// TIA Portal project "A180648-11总成异响" (V14)

(* hardware
DEVICE "S7-1200 station_1"  S7-1200 Station
   slot 0: "Rack_0"  S7-1200 Rack  Rack  V1.0
   slot 1: "A170648_14 CPU  1214C"  CPU 1214C DC/DC/DC  6ES7 214-1AG40-0XB0  V4.2
   slot 2: "DI 16/DQ 16x24VDC_1"  6ES7 223-1BL32-0XB0  V2.0
DEVICE "GSD device_1"  GSD.Device.PN
   slot 0: "机架"  Rack  V1.0
   slot 0: "cv-x100"  CV-X1XX  CV-X1XX  2.0
      slot 0: "CV-X1XX"  CV-X1XX  2.0
      slot 1: "Interface"  Interface
         slot 1: "Port 1"  Port 1
   slot 1: "Command and Result Status_1"  Command and Result Status
      slot 0: "Command and Result Status"  Command and Result Status
   slot 2: "Trg Ready Status_1"  Trg Ready Status
      slot 0: "Trg Ready Status"  Trg Ready Status
   slot 3: "Trg Ack Status_1"  Trg Ack Status
      slot 0: "Trg Ack Status"  Trg Ack Status
   slot 4: "Miscellaneous Status_1"  Miscellaneous Status
      slot 0: "Miscellaneous Status"  Miscellaneous Status
   slot 5: "Tool Judge Value_1"  Tool Judge Value
      slot 0: "Tool Judge Value"  Tool Judge Value
   slot 6: "Result Data 128Byte_1"  Result Data 128Byte
      slot 0: "Result Data 128Byte"  Result Data 128Byte
   slot 7: "Result Data 32Byte_1"  Result Data 32Byte
      slot 0: "Result Data 32Byte"  Result Data 32Byte
   slot 8: "Result Data 32Byte_2"  Result Data 32Byte
      slot 0: "Result Data 32Byte"  Result Data 32Byte
   slot 9: "Result Data 32Byte_3"  Result Data 32Byte
      slot 0: "Result Data 32Byte"  Result Data 32Byte
   slot 10: "Result Data 32Byte_4"  Result Data 32Byte
      slot 0: "Result Data 32Byte"  Result Data 32Byte
   slot 11: "Result Data 32Byte_5"  Result Data 32Byte
      slot 0: "Result Data 32Byte"  Result Data 32Byte
   slot 12: "Command and Result Control_1"  Command and Result Control
      slot 0: "Command and Result Control"  Command and Result Control
   slot 13: "Trg Control_1"  Trg Control
      slot 0: "Trg Control"  Trg Control
   slot 14: "Miscellaneous Control_1"  Miscellaneous Control
      slot 0: "Miscellaneous Control"  Miscellaneous Control
   slot 15: "Reserved Control_1"  Reserved Control
      slot 0: "Reserved Control"  Reserved Control
   slot 16: "Reserved Control_2"  Reserved Control
      slot 0: "Reserved Control"  Reserved Control
   slot 17: "Parameter 128Byte_1"  Parameter 128Byte
      slot 0: "Parameter 128Byte"  Parameter 128Byte
   slot 18: "Parameter 32Byte_1"  Parameter 32Byte
      slot 0: "Parameter 32Byte"  Parameter 32Byte
   slot 19: "Parameter 32Byte_2"  Parameter 32Byte
      slot 0: "Parameter 32Byte"  Parameter 32Byte
   slot 20: "Parameter 32Byte_3"  Parameter 32Byte
      slot 0: "Parameter 32Byte"  Parameter 32Byte
   slot 21: "Parameter 32Byte_4"  Parameter 32Byte
      slot 0: "Parameter 32Byte"  Parameter 32Byte
   slot 22: "Parameter 32Byte_5"  Parameter 32Byte
      slot 0: "Parameter 32Byte"  Parameter 32Byte
*)

// ===== PLC "A170648_14 CPU  1214C"  CPU 1214C DC/DC/DC =====

VAR_GLOBAL   // PLC tag table "默认变量表"
   "启动拍照" AT %I0.0 : Bool;
   "不" AT %I0.1 : Bool;
   "复位" AT %I0.2 : Bool;
   "急停" AT %I0.3 : Bool;
   "Tag_18" AT %IW64 : Int;
   "CMD_complete" AT %I504.0 : Bool;
   "TRG1_feed" AT %I506.0 : Bool;
   "TRG2_feed" AT %I506.1 : Bool;
   "CCD_busy" AT %I507.0 : Bool;
   "CCD_TRG1_NG" AT %I508.0 : Bool;
   "CCD_TRG1_OK" AT %I508.1 : Bool;
   "Conmmad Result" AT %ID588 : DWord;
   "Conmmad Data1" AT %ID592 : DWord;
   "Conmmad Data2" AT %ID596 : DWord;
   "电机拧紧确认" AT %I0.4 : Bool;
   "电机螺栓色标" AT %I3.7 : Bool;
   "电机扎带拾取" AT %I1.1 : Bool;
   "电机扫码启动" AT %I1.2 : Bool;
   "控制器扫码启动" AT %I2.0 : Bool;
   "拧紧枪2确认" AT %I0.5 : Bool;
   "拧紧枪3" AT %I0.6 : Bool;
   "ECU记号笔" AT %I1.5 : Bool;
   "左线卡" AT %I2.2 : Bool;
   "左轧带" AT %I2.5 : Bool;
   "Tag_27" AT %I0.7 : Bool;
   "中轧带" AT %I2.3 : Bool;
   "弹簧取料" AT %I2.4 : Bool;
   "红" AT %Q2.4 : Bool;
   "Tag_17" AT %QW80 : Int;
   "Tag_21" AT %Q3.2 : Bool;
   "Cmd Command" AT %Q504.0 : Bool;
   "CCD_reset" AT %Q504.4 : Bool;
   "TRG1.OUT" AT %Q505.0 : Bool;
   "TRG2.OUT" AT %Q505.1 : Bool;
   "RESET.OUT" AT %Q506.0 : Bool;
   "Tag_65" AT %Q506.1 : Bool;
   "Command NO.OUT" AT %QD580 : DWord;
   "Cmd Parameter1.OUT" AT %QD584 : DWord;
   "Cmd Parameter2.OUT" AT %QD588 : DWord;
   "Cmd Parameter3.OUT" AT %QD592 : DWord;
   "Cmd Parameter4.OUT" AT %QD596 : DWord;
   "Cmd Parameter5.OUT" AT %QD600 : DWord;
   "蜂鸣器" AT %Q2.3 : Bool;
   "Tag_42" AT %Q2.5 : Bool;
   "Tag_43" AT %Q2.6 : Bool;
   "Tag_44" AT %Q2.2 : Bool;
   "安装弹簧" AT %Q20.0 : Bool;
   "安装O型圈" AT %Q20.1 : Bool;
   "安装弹性垫圈弹簧" AT %Q20.2 : Bool;
   "电机安装螺栓1" AT %Q20.3 : Bool;
   "电机安装螺栓2" AT %Q20.4 : Bool;
   "电机安装螺栓3" AT %Q20.5 : Bool;
   "电机拍照" AT %Q20.6 : Bool;
   "涂色标" AT %Q20.7 : Bool;
   "安装轧带取走工" AT %Q21.0 : Bool;
   "Q29" AT %Q21.1 : Bool;
   "Q30" AT %Q21.2 : Bool;
   "Q31" AT %Q21.3 : Bool;
   "Q32" AT %Q21.4 : Bool;
   "Q33" AT %Q21.5 : Bool;
   "Q34" AT %Q21.6 : Bool;
   "Q35" AT %Q21.7 : Bool;
   "程序停止" AT %M100.0 : Bool;
   "复位完成" AT %M100.1 : Bool;
   "Clock_1Hz" AT %M0.5 : Bool;
   "AlwaysFALSE" AT %M1.3 : Bool;
   "Clock_Byte" AT %MB0 : Byte;
   "Clock_10Hz" AT %M0.0 : Bool;
   "Clock_5Hz" AT %M0.1 : Bool;
   "Clock_2.5Hz" AT %M0.2 : Bool;
   "Clock_2Hz" AT %M0.3 : Bool;
   "Clock_1.25Hz" AT %M0.4 : Bool;
   "Clock_0.625Hz" AT %M0.6 : Bool;
   "Clock_0.5Hz" AT %M0.7 : Bool;
   "System_Byte" AT %MB1 : Byte;
   "FirstScan" AT %M1.0 : Bool;
   "DiagStatusUpdate" AT %M1.1 : Bool;
   "AlwaysTRUE" AT %M1.2 : Bool;
   "Tag_19" AT %MD200 : Real;
   "Tag_20" AT %MD204 : Real;
   "磁粉离合器校准" AT %M160.0 : Bool;
   "Tag_22" AT %M300.1 : Bool;
   "Tag_23" AT %M300.2 : Bool;
   "Tag_24" AT %M300.3 : Bool;
   "Tag_25" AT %MW200 : Int;
   "Tag_26" AT %M400.0 : Bool;
   "Tag_1" AT %M200.0 : Bool;
   "Tag_2" AT %M200.1 : Bool;
   "Tag_3" AT %M200.2 : Bool;
   "Tag_4" AT %M200.3 : Bool;
   "Tag_5" AT %M200.4 : Bool;
   "Tag_6" AT %M200.5 : Bool;
   "Tag_7" AT %M200.6 : Bool;
   "Tag_8" AT %M200.7 : Bool;
   "Tag_9" AT %M201.0 : Bool;
   "Tag_10" AT %M201.1 : Bool;
   "Tag_11" AT %M201.2 : Bool;
   "Tag_12" AT %M201.3 : Bool;
   "Tag_13" AT %M201.4 : Bool;
   "Tag_14" AT %M201.5 : Bool;
   "Tag_15" AT %M201.6 : Bool;
   "Tag_16" AT %M201.7 : Bool;
   "Tag_17(1)" AT %M202.0 : Bool;
   "Tag_18(1)" AT %M202.1 : Bool;
   "Tag_19(1)" AT %M202.2 : Bool;
   "Tag_20(1)" AT %M202.3 : Bool;
   "Tag_21(1)" AT %M202.4 : Bool;
   "Tag_22(1)" AT %M202.5 : Bool;
   "Tag_23(1)" AT %M202.6 : Bool;
   "Tag_24(1)" AT %M202.7 : Bool;
   "Tag_37" AT %M203.0 : Bool;
   "Tag_38" AT %M203.1 : Bool;
   "Tag_39" AT %M203.2 : Bool;
   "Tag_40" AT %M205.0 : Bool;
   "Tag_41" AT %M205.1 : Bool;
   "Tag_45" AT %MW600 : Int;
   "Tag_46" AT %M500.0 : Bool;
   "Tag_47" AT %M500.1 : Bool;
   "Tag_48" AT %MW604 : Word;
   "Tag_49" AT %MW608 : Int;
   "Tag_28" AT %M500.3 : Bool;
   "Tag_29" AT %M500.5 : Bool;
   "Tag_30" AT %M501.0 : Bool;
   "Tag_31" AT %M501.1 : Bool;
   "Tag_32" AT %M503.0 : Bool;
   "Tag_33" AT %M503.1 : Bool;
   "Tag_34" AT %M503.2 : Bool;
   "Tag_35" AT %M503.3 : Bool;
   "Tag_36" AT %M503.4 : Bool;
   "Tag_50" AT %M503.5 : Bool;
   "Tag_51" AT %M505.0 : Bool;
   "Tag_52" AT %M506.0 : Bool;
   "Tag_53" AT %M506.1 : Bool;
   "Tag_54" AT %M506.2 : Bool;
   "Tag_55" AT %M506.5 : Bool;
   "Tag_56" AT %M506.6 : Bool;
   "Tag_57" AT %M507.1 : Bool;
   "Tag_58" AT %M507.0 : Bool;
   "Tag_59" AT %M507.2 : Bool;
   "控制器安装螺栓1" AT %Q30.0 : Bool;
   "控制器安装螺栓2" AT %Q30.1 : Bool;
   "控制器安装螺栓3" AT %Q30.2 : Bool;
   "安装支架螺栓1" AT %Q30.3 : Bool;
   "安装支架螺栓2" AT %Q30.4 : Bool;
   "安装支架螺栓3" AT %Q30.5 : Bool;
   "安装支架螺栓4" AT %Q30.6 : Bool;
   "安装支架涂色标" AT %Q30.7 : Bool;
   "安装轧带取走工件" AT %Q31.0 : Bool;
   "备用" AT %Q31.1 : Bool;
   "备用_1" AT %Q31.2 : Bool;
   "备用_2" AT %Q31.3 : Bool;
   "备用_3" AT %Q31.4 : Bool;
   "备用_4" AT %Q31.5 : Bool;
   "备用_5" AT %Q31.6 : Bool;
   "备用_6" AT %Q31.7 : Bool;
   "Tag_60" AT %M507.3 : Bool;
   "Tag_61" AT %M507.4 : Bool;
   "Tag_62" AT %M507.5 : Bool;
   "Tag_63" AT %M507.6 : Bool;
   "Tag_64" AT %M507.7 : Bool;
   "Tag_66" AT %M508.0 : Bool;
   "Tag_67" AT %M508.1 : Bool;
   "Tag_68" AT %M508.2 : Bool;
   "Tag_69" AT %M508.3 : Bool;
   "Tag_70" AT %M508.4 : Bool;
   "Tag_71" AT %M508.5 : Bool;
   "Tag_72" AT %M508.6 : Bool;
   "Tag_73" AT %M508.7 : Bool;
END_VAR

DATA_BLOCK "SERVER"   // DB1
{ S7_Optimized_Access := 'FALSE' }
VERSION : 0.1
   VAR
      设备状态1 : Int := 0;
      设备状态2 : Int;
      设备状态3 : Int;
      产品型号 : Int := 0;
      错误代码 : Int := 0;
      生产结果 : Int := 0;
      设备编号 : Int := 0;
      产品标识 : Int;
      胶垫弹簧CCD程序号 : Int;
      电机方向程序号 : Int;
      电机螺栓数量 : Int;
      合装螺栓1数量 : Int;
      合装螺栓2数量 : Int;
      控制器螺栓数量 : Int;
      ECU安装 : Array[0..16] of Bool;
   END_VAR
BEGIN
END_DATA_BLOCK

DATA_BLOCK "MB_TCON"   // DB2
{ S7_Optimized_Access := 'FALSE' }
VERSION : 0.1
   VAR
      MB_TCON : TCON_IP_v4;
   END_VAR
BEGIN
   MB_TCON.InterfaceId := 64;
   MB_TCON.ID := 1;
   MB_TCON.LocalPort := 502;
   MB_TCON.RemoteAddress.ADDR[1] := 0;
   MB_TCON.RemoteAddress.ADDR[2] := 0;
   MB_TCON.RemoteAddress.ADDR[3] := 0;
   MB_TCON.RemoteAddress.ADDR[4] := 0;
END_DATA_BLOCK

DATA_BLOCK "RESET_DB"   // DB3
{ S7_Optimized_Access := 'TRUE' }
VERSION : 0.1
// stored: InstanceOfName RESET
"RESET"
BEGIN
END_DATA_BLOCK

DATA_BLOCK "ALARM_DB"   // DB4
{ S7_Optimized_Access := 'TRUE' }
VERSION : 0.1
// stored: InstanceOfName ALARM
"ALARM"
BEGIN
END_DATA_BLOCK

DATA_BLOCK "CCD检测_DB"   // DB6
{ S7_Optimized_Access := 'TRUE' }
VERSION : 0.1
// stored: InstanceOfName CCD检测
"CCD检测"
BEGIN
END_DATA_BLOCK

DATA_BLOCK "AUTO_DB"   // DB10
{ S7_Optimized_Access := 'TRUE' }
VERSION : 0.1
// stored: InstanceOfName AUTO
"AUTO"
BEGIN
END_DATA_BLOCK

// folder: System blocks/Program resources

DATA_BLOCK "IEC_Timer_0_DB"   // DB5
{ S7_Optimized_Access := 'TRUE' }
AUTHOR : Simatic
FAMILY : IEC
NAME : IEC_TMR
VERSION : 1.0
// stored: InstanceOfName IEC_TIMER
"IEC_TIMER"
BEGIN
END_DATA_BLOCK

DATA_BLOCK "IEC_Timer_0_DB_3"   // DB12
{ S7_Optimized_Access := 'TRUE' }
AUTHOR : Simatic
FAMILY : IEC
NAME : IEC_TMR
VERSION : 1.0
// stored: InstanceOfName IEC_TIMER
"IEC_TIMER"
BEGIN
END_DATA_BLOCK

// folder: (top level)

FUNCTION_BLOCK "ALARM"   // FB1, LAD
{ S7_Optimized_Access := 'TRUE' }
VERSION : 0.1
   VAR
      "Error-ID" : Word;
      TEmp : Array[0..3] of Bool;
      IEC_Timer_0_Instance : TON_TIME;
      IEC_Timer_0_Instance_1 : TON_TIME;
      IEC_Timer_0_Instance_2 : TON_TIME;
      IEC_Timer_0_Instance_3 : TON_TIME;
      IEC_Timer_0_Instance_4 : TON_TIME;
      IEC_Timer_0_Instance_5 : TON_TIME;
      IEC_Timer_0_Instance_6 : TON_TIME;
      IEC_Timer_0_Instance_7 : TON_TIME;
      IEC_Timer_0_Instance_8 : TON_TIME;
      IEC_Timer_0_Instance_9 : TON_TIME;
      IEC_Timer_0_Instance_10 : TON_TIME;
      IEC_Timer_0_Instance_11 : TON_TIME;
      IEC_Timer_0_Instance_12 : TON_TIME;
      IEC_Timer_0_Instance_13 : TON_TIME;
      IEC_Timer_0_Instance_14 : TON_TIME;
      "STEP" : Int;
      IEC_Timer_0_Instance_15 : TON_TIME;
      IEC_Timer_0_Instance_16 : TON_TIME;
   END_VAR
BEGIN

REGION Network 1
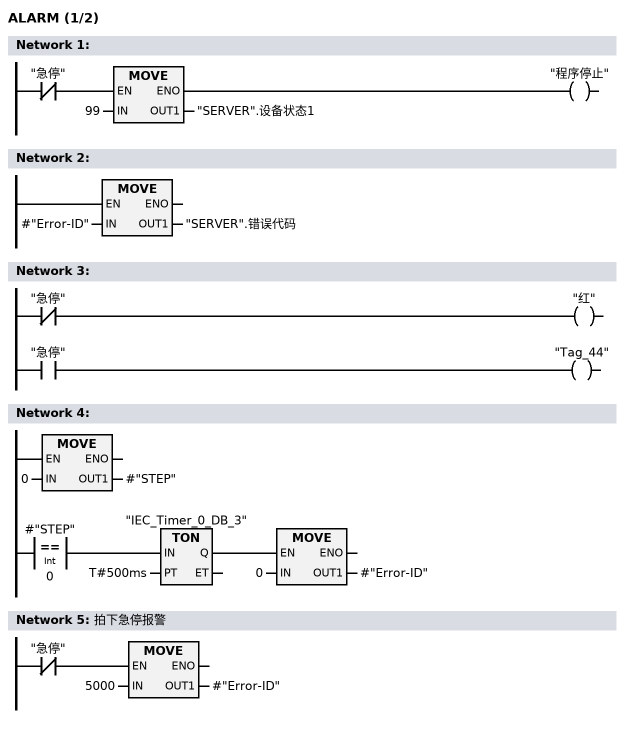
   RUNG wire#powerrail
      I_Contact( "急停" )
      Move(in := 99, out1 => "SERVER".设备状态1)
      Coil( "程序停止" )
   END_RUNG
   // the same network as SCL:
   IF NOT "急停" THEN "SERVER".设备状态1 := 99; END_IF;
   "程序停止" := NOT "急停";
END_REGION

REGION Network 2
   RUNG wire#powerrail
      Move(in := #"Error-ID", out1 => "SERVER".错误代码)
   END_RUNG
   // the same network as SCL:
   "SERVER".错误代码 := #"Error-ID";
END_REGION

REGION Network 3
   RUNG wire#powerrail
      I_Contact( "急停" )
      Coil( "红" )
   END_RUNG
   RUNG wire#powerrail
      Contact( "急停" )
      Coil( "Tag_44" )
   END_RUNG
   // the same network as SCL:
   "红" := NOT "急停";
   "Tag_44" := "急停";
END_REGION

REGION Network 4
   #"STEP" := 0;
   "IEC_Timer_0_DB_3".TON(IN := #"STEP" = 0, PT := T#500ms);
   IF "IEC_Timer_0_DB_3".Q THEN #"Error-ID" := 0; END_IF;
END_REGION

REGION Network 5: 拍下急停报警
   RUNG wire#powerrail
      I_Contact( "急停" )
      Move(in := 5000, out1 => #"Error-ID")
   END_RUNG
   // the same network as SCL:
   IF NOT "急停" THEN #"Error-ID" := 5000; END_IF;
END_REGION

REGION Network 6: 安全门打开报警
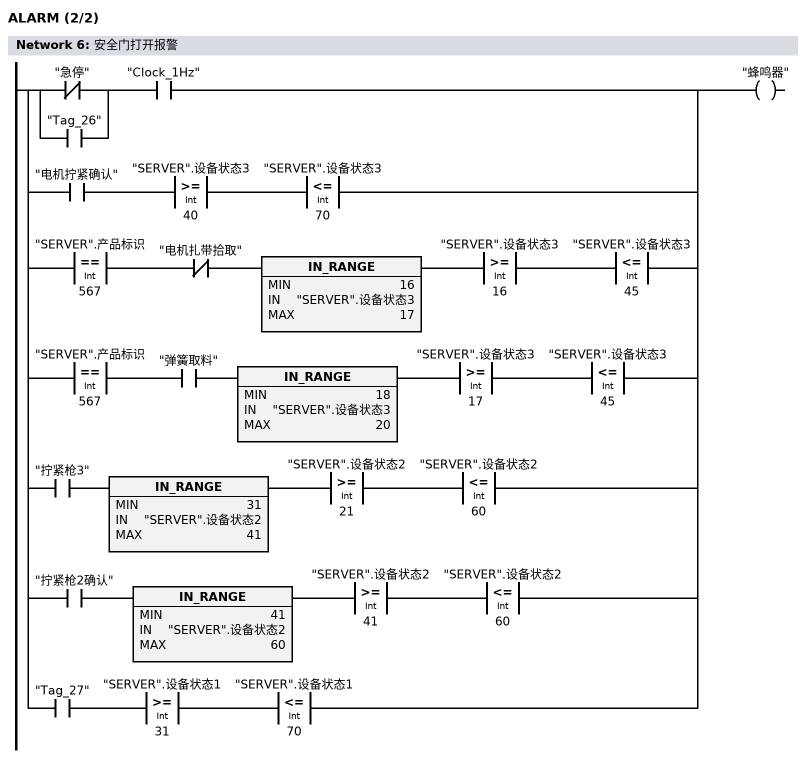
   RUNG wire#powerrail
      I_Contact( "急停" )
      wire#w1
      Contact( "Clock_1Hz" )
      wire#w2
      Coil( "蜂鸣器" )
   END_RUNG
   RUNG wire#powerrail
      Contact( "Tag_26" )
   END_RUNG wire#w1
   RUNG wire#powerrail
      Contact( "电机拧紧确认" )
      { S7_Templates := "SrcType := Int" } GE_Contact(in1 := "SERVER".设备状态3, in2 := 40)
      { S7_Templates := "SrcType := Int" } LE_Contact(in1 := "SERVER".设备状态3, in2 := 70)
   END_RUNG wire#w2
   RUNG wire#powerrail
      { S7_Templates := "SrcType := Int" } EQ_Contact(in1 := "SERVER".产品标识, in2 := 567)
      I_Contact( "电机扎带拾取" )
      { S7_Templates := "SrcType := Int" } InRange(min := 16, in := "SERVER".设备状态3, max := 17)
      { S7_Templates := "SrcType := Int" } GE_Contact(in1 := "SERVER".设备状态3, in2 := 16)
      { S7_Templates := "SrcType := Int" } LE_Contact(in1 := "SERVER".设备状态3, in2 := 45)
   END_RUNG wire#w2
   RUNG wire#powerrail
      { S7_Templates := "SrcType := Int" } EQ_Contact(in1 := "SERVER".产品标识, in2 := 567)
      Contact( "弹簧取料" )
      { S7_Templates := "SrcType := Int" } InRange(min := 18, in := "SERVER".设备状态3, max := 20)
      { S7_Templates := "SrcType := Int" } GE_Contact(in1 := "SERVER".设备状态3, in2 := 17)
      { S7_Templates := "SrcType := Int" } LE_Contact(in1 := "SERVER".设备状态3, in2 := 45)
   END_RUNG wire#w2
   RUNG wire#powerrail
      Contact( "拧紧枪3" )
      { S7_Templates := "SrcType := Int" } InRange(min := 31, in := "SERVER".设备状态2, max := 41)
      { S7_Templates := "SrcType := Int" } GE_Contact(in1 := "SERVER".设备状态2, in2 := 21)
      { S7_Templates := "SrcType := Int" } LE_Contact(in1 := "SERVER".设备状态2, in2 := 60)
   END_RUNG wire#w2
   RUNG wire#powerrail
      Contact( "拧紧枪2确认" )
      { S7_Templates := "SrcType := Int" } InRange(min := 41, in := "SERVER".设备状态2, max := 60)
      { S7_Templates := "SrcType := Int" } GE_Contact(in1 := "SERVER".设备状态2, in2 := 41)
      { S7_Templates := "SrcType := Int" } LE_Contact(in1 := "SERVER".设备状态2, in2 := 60)
   END_RUNG wire#w2
   RUNG wire#powerrail
      Contact( "Tag_27" )
      { S7_Templates := "SrcType := Int" } GE_Contact(in1 := "SERVER".设备状态1, in2 := 31)
      { S7_Templates := "SrcType := Int" } LE_Contact(in1 := "SERVER".设备状态1, in2 := 70)
   END_RUNG wire#w2
   // the same network as SCL:
   "蜂鸣器" := ((NOT "急停" OR "Tag_26") AND "Clock_1Hz") OR ("电机拧紧确认" AND ("SERVER".设备状态3 >= 40) AND ("SERVER".设备状态3 <= 70)) OR (("SERVER".产品标识 = 567) AND NOT "电机扎带拾取" AND (16 <= "SERVER".设备状态3) AND ("SERVER".设备状态3 <= 17) AND ("SERVER".设备状态3 >= 16) AND ("SERVER".设备状态3 <= 45)) OR (("SERVER".产品标识 = 567) AND "弹簧取料" AND (18 <= "SERVER".设备状态3) AND ("SERVER".设备状态3 <= 20) AND ("SERVER".设备状态3 >= 17) AND ("SERVER".设备状态3 <= 45)) OR ("拧紧枪3" AND (31 <= "SERVER".设备状态2) AND ("SERVER".设备状态2 <= 41) AND ("SERVER".设备状态2 >= 21) AND ("SERVER".设备状态2 <= 60)) OR ("拧紧枪2确认" AND (41 <= "SERVER".设备状态2) AND ("SERVER".设备状态2 <= 60) AND ("SERVER".设备状态2 >= 41) AND ("SERVER".设备状态2 <= 60)) OR ("Tag_27" AND ("SERVER".设备状态1 >= 31) AND ("SERVER".设备状态1 <= 70));
END_REGION

REGION Network 7: 工件未在位启动报警
END_REGION

REGION Network 8: 气源未开报警
END_REGION

REGION Network 9: 工装移栽前进未到位报警
END_REGION

REGION Network 10: 工装移栽未后退报警
END_REGION

REGION Network 11: 防护门未上升报警
END_REGION

REGION Network 12: 防护门为下降报警
END_REGION

REGION Network 13: 1#固定气缸未锁紧报警
END_REGION

REGION Network 14: 1#固定气缸未退回报警
END_REGION

REGION Network 15: 1#机械手未上升报警
END_REGION

REGION Network 16: 1#机械手未下降报警
END_REGION

REGION Network 17: 1#气爪未夹紧到位报警
END_REGION

REGION Network 18: 1#气爪未松开报警
END_REGION

REGION Network 19: 2#机械手未固定锁紧报警
END_REGION

REGION Network 20: 2#固定气缸未退回报警
END_REGION

REGION Network 21: 2#机械手未上升报警
END_REGION

REGION Network 22: 2#机械手未下降报警
END_REGION

REGION Network 23: 2#气爪未夹紧报警
END_REGION

REGION Network 24: 2#气爪未松开报警
END_REGION

REGION Network 25: 激光打码报警
END_REGION
END_FUNCTION_BLOCK

FUNCTION_BLOCK "RESET"   // FB2, LAD
{ S7_Optimized_Access := 'TRUE' }
VERSION : 0.1
   VAR_INPUT
      Stop : Bool;
      Start : Bool;
   END_VAR
   VAR_OUTPUT
      Down : Bool;
   END_VAR
   VAR
      "Step" : Int;
   END_VAR
BEGIN

REGION Network 1
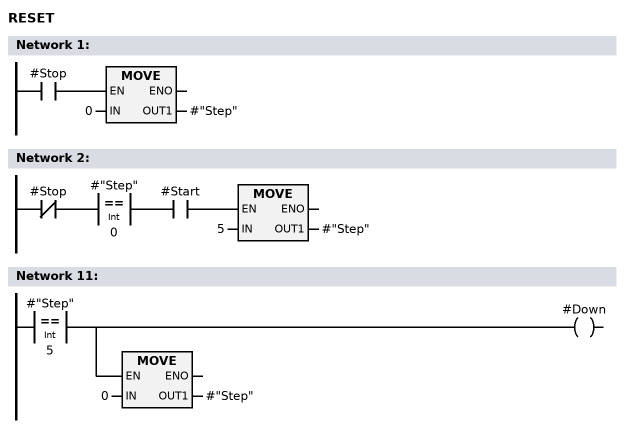
   RUNG wire#powerrail
      Contact( #Stop )
      Move(in := 0, out1 => #"Step")
   END_RUNG
   // the same network as SCL:
   IF #Stop THEN #"Step" := 0; END_IF;
END_REGION

REGION Network 2
   RUNG wire#powerrail
      I_Contact( #Stop )
      { S7_Templates := "SrcType := Int" } EQ_Contact(in1 := #"Step", in2 := 0)
      Contact( #Start )
      Move(in := 5, out1 => #"Step")
   END_RUNG
   // the same network as SCL:
   IF NOT #Stop AND (#"Step" = 0) AND #Start THEN #"Step" := 5; END_IF;
END_REGION

REGION Network 7: 1#气爪松开
END_REGION

REGION Network 8: 2#气爪松开
END_REGION

REGION Network 11
   RUNG wire#powerrail
      { S7_Templates := "SrcType := Int" } EQ_Contact(in1 := #"Step", in2 := 5)
      wire#w1
      Coil( #Down )
   END_RUNG
   RUNG wire#w1
      Move(in := 0, out1 => #"Step")
   END_RUNG
   // the same network as SCL:
   #Down := #"Step" = 5;
   IF #Down THEN #"Step" := 0; END_IF;
END_REGION
END_FUNCTION_BLOCK

FUNCTION_BLOCK "AUTO"   // FB3, LAD
{ S7_Optimized_Access := 'TRUE' }
VERSION : 0.1
   VAR
      IEC_Timer_0_Instance : TON_TIME;
      IEC_Timer_0_Instance_1 : TON_TIME;
      IEC_Timer_0_Instance_2 : TON_TIME;
      IEC_Timer_0_Instance_3 : TON_TIME;
      IEC_Timer_0_Instance_4 : TON_TIME;
      IEC_Timer_0_Instance_5 : TON_TIME;
      IEC_Timer_0_Instance_6 : TON_TIME;
      IEC_Timer_0_Instance_7 : TON_TIME;
      IEC_Timer_0_Instance_8 : TON_TIME;
      IEC_Timer_0_Instance_9 : TON_TIME;
      IEC_Timer_0_Instance_10 : TON_TIME;
      IEC_Timer_0_Instance_11 : TON_TIME;
      IEC_Timer_0_Instance_12 : TON_TIME;
      IEC_Timer_0_Instance_13 : TON_TIME;
      IEC_Timer_0_Instance_14 : TON_TIME;
      IEC_Timer_0_Instance_15 : TON_TIME;
      IEC_Timer_0_Instance_16 : TON_TIME;
      IEC_Timer_0_Instance_17 : TON_TIME;
      IEC_Timer_0_Instance_18 : TON_TIME;
      IEC_Timer_0_Instance_19 : TON_TIME;
      IEC_Timer_0_Instance_20 : TON_TIME;
      IEC_Timer_0_Instance_22 : TON_TIME;
      IEC_Timer_0_Instance_23 : TON_TIME;
      IEC_Timer_0_Instance_21 : TON_TIME;
   END_VAR
   VAR_TEMP
      temp0 : Bool;
      temp1 : Bool;
      temp2 : Bool;
      temp17 : Bool;
      temp4 : Bool;
      temp5 : Bool;
      temp6 : Bool;
      temp7 : Bool;
      temp8 : Bool;
      temp9 : Bool;
      temp10 : Bool;
      temp11 : Bool;
      temp12 : Bool;
      temp13 : Bool;
      temp14 : Bool;
      temp15 : Bool;
      temp16 : Bool;
      temp18 : Bool;
      temp19 : Bool;
      temp20 : Bool;
      temp21 : Bool;
   END_VAR
   VAR_TEMP   // added for the SCL form of the ladder/FBD networks
      _w1 : Bool;
      _w2 : Bool;
      _w3 : Bool;
      _w4 : Bool;
   END_VAR
BEGIN

REGION Network 1
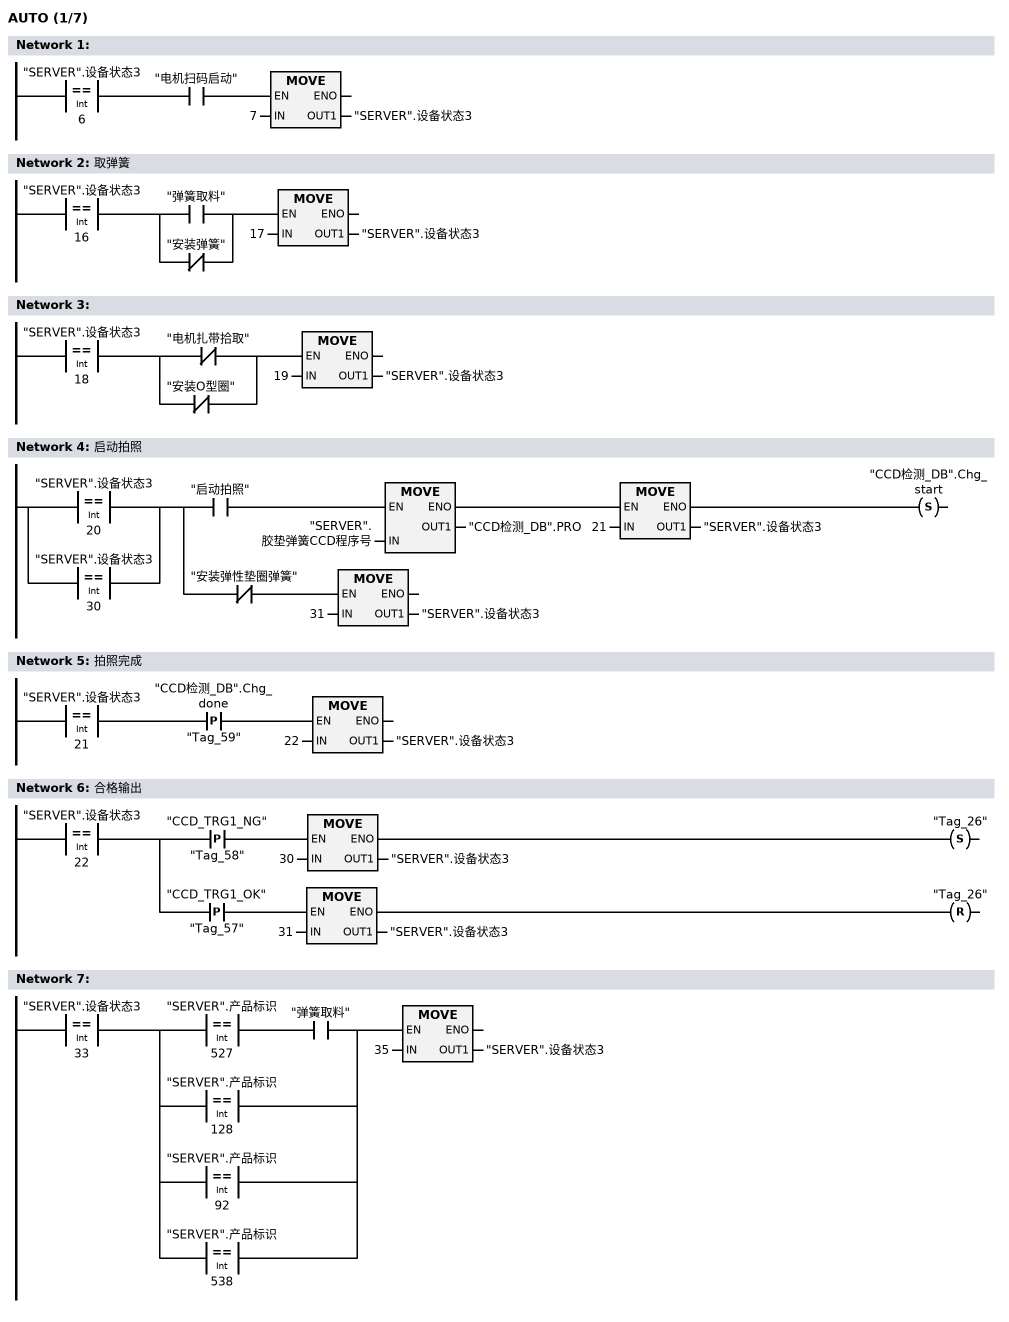
   RUNG wire#powerrail
      { S7_Templates := "SrcType := Int" } EQ_Contact(in1 := "SERVER".设备状态3, in2 := 6)
      Contact( "电机扫码启动" )
      Move(in := 7, out1 => "SERVER".设备状态3)
   END_RUNG
   // the same network as SCL:
   IF ("SERVER".设备状态3 = 6) AND "电机扫码启动" THEN "SERVER".设备状态3 := 7; END_IF;
END_REGION

REGION Network 2: 取弹簧
   RUNG wire#powerrail
      { S7_Templates := "SrcType := Int" } EQ_Contact(in1 := "SERVER".设备状态3, in2 := 16)
      wire#w1
      Contact( "弹簧取料" )
      wire#w2
      Move(in := 17, out1 => "SERVER".设备状态3)
   END_RUNG
   RUNG wire#w1
      I_Contact( "安装弹簧" )
   END_RUNG wire#w2
   // the same network as SCL:
   IF ("SERVER".设备状态3 = 16) AND ("弹簧取料" OR NOT "安装弹簧") THEN "SERVER".设备状态3 := 17; END_IF;
END_REGION

REGION Network 3
   RUNG wire#powerrail
      { S7_Templates := "SrcType := Int" } EQ_Contact(in1 := "SERVER".设备状态3, in2 := 18)
      wire#w1
      I_Contact( "电机扎带拾取" )
      wire#w2
      Move(in := 19, out1 => "SERVER".设备状态3)
   END_RUNG
   RUNG wire#w1
      I_Contact( "安装O型圈" )
   END_RUNG wire#w2
   // the same network as SCL:
   IF ("SERVER".设备状态3 = 18) AND (NOT "电机扎带拾取" OR NOT "安装O型圈") THEN "SERVER".设备状态3 := 19; END_IF;
END_REGION

REGION Network 4: 启动拍照
   RUNG wire#powerrail
      { S7_Templates := "SrcType := Int" } EQ_Contact(in1 := "SERVER".设备状态3, in2 := 20)
      wire#w1
      Contact( "启动拍照" )
      Move(in := "SERVER".胶垫弹簧CCD程序号, out1 => "CCD检测_DB".PRO)
      Move(in := 21, out1 => "SERVER".设备状态3)
      S_Coil( "CCD检测_DB".Chg_start )
   END_RUNG
   RUNG wire#powerrail
      { S7_Templates := "SrcType := Int" } EQ_Contact(in1 := "SERVER".设备状态3, in2 := 30)
   END_RUNG wire#w1
   RUNG wire#w1
      I_Contact( "安装弹性垫圈弹簧" )
      Move(in := 31, out1 => "SERVER".设备状态3)
   END_RUNG
   // the same network as SCL:
   #_w1 := ("SERVER".设备状态3 = 20) OR ("SERVER".设备状态3 = 30);
   IF #_w1 AND "启动拍照" THEN
       "CCD检测_DB".PRO := "SERVER".胶垫弹簧CCD程序号;
       "SERVER".设备状态3 := 21;
       "CCD检测_DB".Chg_start := TRUE;
   END_IF;
   IF #_w1 AND NOT "安装弹性垫圈弹簧" THEN "SERVER".设备状态3 := 31; END_IF;
END_REGION

REGION Network 5: 拍照完成
   RUNG wire#powerrail
      { S7_Templates := "SrcType := Int" } EQ_Contact(in1 := "SERVER".设备状态3, in2 := 21)
      P_Contact(operand := "CCD检测_DB".Chg_done, bit := "Tag_59")
      Move(in := 22, out1 => "SERVER".设备状态3)
   END_RUNG
   // the same network as SCL:
   #_w1 := ("SERVER".设备状态3 = 21) AND "CCD检测_DB".Chg_done AND NOT "Tag_59";   // rising edge of "CCD检测_DB".Chg_done
   "Tag_59" := "CCD检测_DB".Chg_done;
   IF #_w1 THEN "SERVER".设备状态3 := 22; END_IF;
END_REGION

REGION Network 6: 合格输出
   RUNG wire#powerrail
      { S7_Templates := "SrcType := Int" } EQ_Contact(in1 := "SERVER".设备状态3, in2 := 22)
      wire#w1
      P_Contact(operand := "CCD_TRG1_NG", bit := "Tag_58")
      Move(in := 30, out1 => "SERVER".设备状态3)
      S_Coil( "Tag_26" )
   END_RUNG
   RUNG wire#w1
      P_Contact(operand := "CCD_TRG1_OK", bit := "Tag_57")
      Move(in := 31, out1 => "SERVER".设备状态3)
      R_Coil( "Tag_26" )
   END_RUNG
   // the same network as SCL:
   #_w1 := "SERVER".设备状态3 = 22;
   #_w2 := #_w1 AND "CCD_TRG1_NG" AND NOT "Tag_58";   // rising edge of "CCD_TRG1_NG"
   "Tag_58" := "CCD_TRG1_NG";
   IF #_w2 THEN
       "SERVER".设备状态3 := 30;
       "Tag_26" := TRUE;
   END_IF;
   #_w3 := #_w1 AND "CCD_TRG1_OK" AND NOT "Tag_57";   // rising edge of "CCD_TRG1_OK"
   "Tag_57" := "CCD_TRG1_OK";
   IF #_w3 THEN
       "SERVER".设备状态3 := 31;
       "Tag_26" := FALSE;
   END_IF;
END_REGION

REGION Network 7
   RUNG wire#powerrail
      { S7_Templates := "SrcType := Int" } EQ_Contact(in1 := "SERVER".设备状态3, in2 := 33)
      wire#w1
      { S7_Templates := "SrcType := Int" } EQ_Contact(in1 := "SERVER".产品标识, in2 := 527)
      Contact( "弹簧取料" )
      wire#w2
      Move(in := 35, out1 => "SERVER".设备状态3)
   END_RUNG
   RUNG wire#w1
      { S7_Templates := "SrcType := Int" } EQ_Contact(in1 := "SERVER".产品标识, in2 := 128)
   END_RUNG wire#w2
   RUNG wire#w1
      { S7_Templates := "SrcType := Int" } EQ_Contact(in1 := "SERVER".产品标识, in2 := 92)
   END_RUNG wire#w2
   RUNG wire#w1
      { S7_Templates := "SrcType := Int" } EQ_Contact(in1 := "SERVER".产品标识, in2 := 538)
   END_RUNG wire#w2
   // the same network as SCL:
   IF ("SERVER".设备状态3 = 33) AND ((("SERVER".产品标识 = 527) AND "弹簧取料") OR ("SERVER".产品标识 = 128) OR ("SERVER".产品标识 = 92) OR ("SERVER".产品标识 = 538)) THEN
       "SERVER".设备状态3 := 35;
   END_IF;
END_REGION

REGION Network 8
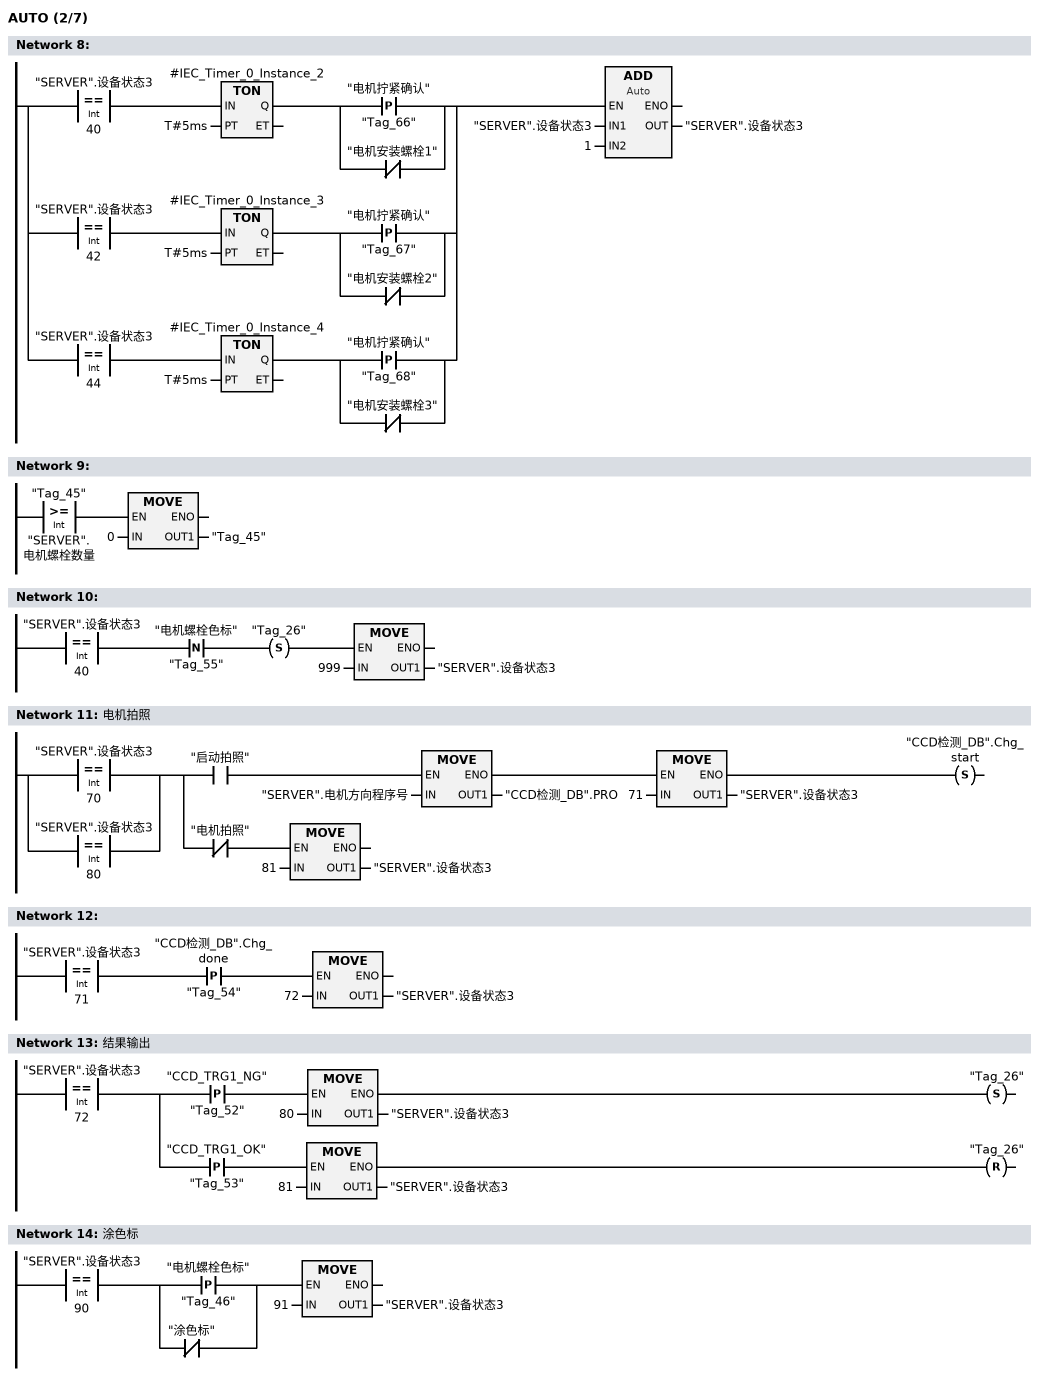
   #IEC_Timer_0_Instance_2(IN := "SERVER".设备状态3 = 40, PT := T#5ms);   // TON
   #_w1 := #IEC_Timer_0_Instance_2.Q AND "电机拧紧确认" AND NOT "Tag_66";   // rising edge of "电机拧紧确认"
   "Tag_66" := "电机拧紧确认";
   #IEC_Timer_0_Instance_3(IN := "SERVER".设备状态3 = 42, PT := T#5ms);   // TON
   #_w2 := #IEC_Timer_0_Instance_3.Q AND "电机拧紧确认" AND NOT "Tag_67";   // rising edge of "电机拧紧确认"
   "Tag_67" := "电机拧紧确认";
   #IEC_Timer_0_Instance_4(IN := "SERVER".设备状态3 = 44, PT := T#5ms);   // TON
   #_w3 := #IEC_Timer_0_Instance_4.Q AND "电机拧紧确认" AND NOT "Tag_68";   // rising edge of "电机拧紧确认"
   "Tag_68" := "电机拧紧确认";
   IF #_w1 OR (#IEC_Timer_0_Instance_2.Q AND NOT "电机安装螺栓1") OR #_w2 OR (#IEC_Timer_0_Instance_3.Q AND NOT "电机安装螺栓2") OR #_w3 OR (#IEC_Timer_0_Instance_4.Q AND NOT "电机安装螺栓3") THEN
       "SERVER".设备状态3 := "SERVER".设备状态3 + 1;
   END_IF;
END_REGION

REGION Network 9
   RUNG wire#powerrail
      { S7_Templates := "SrcType := Int" } GE_Contact(in1 := "Tag_45", in2 := "SERVER".电机螺栓数量)
      Move(in := 0, out1 => "Tag_45")
   END_RUNG
   // the same network as SCL:
   IF "Tag_45" >= "SERVER".电机螺栓数量 THEN "Tag_45" := 0; END_IF;
END_REGION

REGION Network 10
   RUNG wire#powerrail
      { S7_Templates := "SrcType := Int" } EQ_Contact(in1 := "SERVER".设备状态3, in2 := 40)
      N_Contact(operand := "电机螺栓色标", bit := "Tag_55")
      S_Coil( "Tag_26" )
      Move(in := 999, out1 => "SERVER".设备状态3)
   END_RUNG
   // the same network as SCL:
   #_w1 := ("SERVER".设备状态3 = 40) AND NOT "电机螺栓色标" AND "Tag_55";   // falling edge of "电机螺栓色标"
   "Tag_55" := "电机螺栓色标";
   IF #_w1 THEN
       "Tag_26" := TRUE;
       "SERVER".设备状态3 := 999;
   END_IF;
END_REGION

REGION Network 11: 电机拍照
   RUNG wire#powerrail
      { S7_Templates := "SrcType := Int" } EQ_Contact(in1 := "SERVER".设备状态3, in2 := 70)
      wire#w1
      Contact( "启动拍照" )
      Move(in := "SERVER".电机方向程序号, out1 => "CCD检测_DB".PRO)
      Move(in := 71, out1 => "SERVER".设备状态3)
      S_Coil( "CCD检测_DB".Chg_start )
   END_RUNG
   RUNG wire#powerrail
      { S7_Templates := "SrcType := Int" } EQ_Contact(in1 := "SERVER".设备状态3, in2 := 80)
   END_RUNG wire#w1
   RUNG wire#w1
      I_Contact( "电机拍照" )
      Move(in := 81, out1 => "SERVER".设备状态3)
   END_RUNG
   // the same network as SCL:
   #_w1 := ("SERVER".设备状态3 = 70) OR ("SERVER".设备状态3 = 80);
   IF #_w1 AND "启动拍照" THEN
       "CCD检测_DB".PRO := "SERVER".电机方向程序号;
       "SERVER".设备状态3 := 71;
       "CCD检测_DB".Chg_start := TRUE;
   END_IF;
   IF #_w1 AND NOT "电机拍照" THEN "SERVER".设备状态3 := 81; END_IF;
END_REGION

REGION Network 12
   RUNG wire#powerrail
      { S7_Templates := "SrcType := Int" } EQ_Contact(in1 := "SERVER".设备状态3, in2 := 71)
      P_Contact(operand := "CCD检测_DB".Chg_done, bit := "Tag_54")
      Move(in := 72, out1 => "SERVER".设备状态3)
   END_RUNG
   // the same network as SCL:
   #_w1 := ("SERVER".设备状态3 = 71) AND "CCD检测_DB".Chg_done AND NOT "Tag_54";   // rising edge of "CCD检测_DB".Chg_done
   "Tag_54" := "CCD检测_DB".Chg_done;
   IF #_w1 THEN "SERVER".设备状态3 := 72; END_IF;
END_REGION

REGION Network 13: 结果输出
   RUNG wire#powerrail
      { S7_Templates := "SrcType := Int" } EQ_Contact(in1 := "SERVER".设备状态3, in2 := 72)
      wire#w1
      P_Contact(operand := "CCD_TRG1_NG", bit := "Tag_52")
      Move(in := 80, out1 => "SERVER".设备状态3)
      S_Coil( "Tag_26" )
   END_RUNG
   RUNG wire#w1
      P_Contact(operand := "CCD_TRG1_OK", bit := "Tag_53")
      Move(in := 81, out1 => "SERVER".设备状态3)
      R_Coil( "Tag_26" )
   END_RUNG
   // the same network as SCL:
   #_w1 := "SERVER".设备状态3 = 72;
   #_w2 := #_w1 AND "CCD_TRG1_NG" AND NOT "Tag_52";   // rising edge of "CCD_TRG1_NG"
   "Tag_52" := "CCD_TRG1_NG";
   IF #_w2 THEN
       "SERVER".设备状态3 := 80;
       "Tag_26" := TRUE;
   END_IF;
   #_w3 := #_w1 AND "CCD_TRG1_OK" AND NOT "Tag_53";   // rising edge of "CCD_TRG1_OK"
   "Tag_53" := "CCD_TRG1_OK";
   IF #_w3 THEN
       "SERVER".设备状态3 := 81;
       "Tag_26" := FALSE;
   END_IF;
END_REGION

REGION Network 14: 涂色标
   RUNG wire#powerrail
      { S7_Templates := "SrcType := Int" } EQ_Contact(in1 := "SERVER".设备状态3, in2 := 90)
      wire#w1
      P_Contact(operand := "电机螺栓色标", bit := "Tag_46")
      wire#w2
      Move(in := 91, out1 => "SERVER".设备状态3)
   END_RUNG
   RUNG wire#w1
      I_Contact( "涂色标" )
   END_RUNG wire#w2
   // the same network as SCL:
   #_w1 := ("SERVER".设备状态3 = 90) AND "电机螺栓色标" AND NOT "Tag_46";   // rising edge of "电机螺栓色标"
   "Tag_46" := "电机螺栓色标";
   IF #_w1 OR (("SERVER".设备状态3 = 90) AND NOT "涂色标") THEN "SERVER".设备状态3 := 91; END_IF;
END_REGION

REGION Network 15
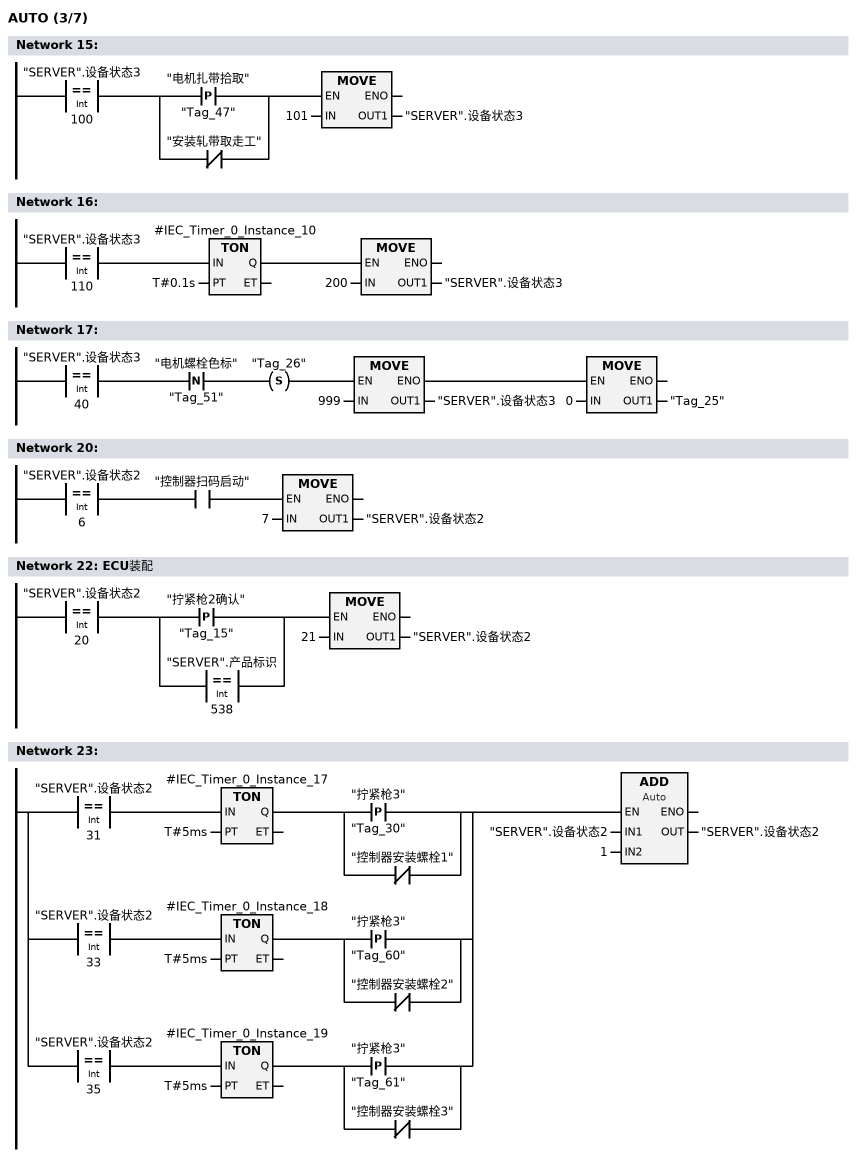
   RUNG wire#powerrail
      { S7_Templates := "SrcType := Int" } EQ_Contact(in1 := "SERVER".设备状态3, in2 := 100)
      wire#w1
      P_Contact(operand := "电机扎带拾取", bit := "Tag_47")
      wire#w2
      Move(in := 101, out1 => "SERVER".设备状态3)
   END_RUNG
   RUNG wire#w1
      I_Contact( "安装轧带取走工" )
   END_RUNG wire#w2
   // the same network as SCL:
   #_w1 := ("SERVER".设备状态3 = 100) AND "电机扎带拾取" AND NOT "Tag_47";   // rising edge of "电机扎带拾取"
   "Tag_47" := "电机扎带拾取";
   IF #_w1 OR (("SERVER".设备状态3 = 100) AND NOT "安装轧带取走工") THEN "SERVER".设备状态3 := 101; END_IF;
END_REGION

REGION Network 16
   #IEC_Timer_0_Instance_10(IN := "SERVER".设备状态3 = 110, PT := T#0.1s);   // TON
   IF #IEC_Timer_0_Instance_10.Q THEN "SERVER".设备状态3 := 200; END_IF;
END_REGION

REGION Network 17
   RUNG wire#powerrail
      { S7_Templates := "SrcType := Int" } EQ_Contact(in1 := "SERVER".设备状态3, in2 := 40)
      N_Contact(operand := "电机螺栓色标", bit := "Tag_51")
      S_Coil( "Tag_26" )
      Move(in := 999, out1 => "SERVER".设备状态3)
      Move(in := 0, out1 => "Tag_25")
   END_RUNG
   // the same network as SCL:
   #_w1 := ("SERVER".设备状态3 = 40) AND NOT "电机螺栓色标" AND "Tag_51";   // falling edge of "电机螺栓色标"
   "Tag_51" := "电机螺栓色标";
   IF #_w1 THEN
       "Tag_26" := TRUE;
       "SERVER".设备状态3 := 999;
       "Tag_25" := 0;
   END_IF;
END_REGION

REGION Network 20
   RUNG wire#powerrail
      { S7_Templates := "SrcType := Int" } EQ_Contact(in1 := "SERVER".设备状态2, in2 := 6)
      Contact( "控制器扫码启动" )
      Move(in := 7, out1 => "SERVER".设备状态2)
   END_RUNG
   // the same network as SCL:
   IF ("SERVER".设备状态2 = 6) AND "控制器扫码启动" THEN "SERVER".设备状态2 := 7; END_IF;
END_REGION

REGION Network 22: ECU装配
   RUNG wire#powerrail
      { S7_Templates := "SrcType := Int" } EQ_Contact(in1 := "SERVER".设备状态2, in2 := 20)
      wire#w1
      P_Contact(operand := "拧紧枪2确认", bit := "Tag_15")
      wire#w2
      Move(in := 21, out1 => "SERVER".设备状态2)
   END_RUNG
   RUNG wire#w1
      { S7_Templates := "SrcType := Int" } EQ_Contact(in1 := "SERVER".产品标识, in2 := 538)
   END_RUNG wire#w2
   // the same network as SCL:
   #_w1 := ("SERVER".设备状态2 = 20) AND "拧紧枪2确认" AND NOT "Tag_15";   // rising edge of "拧紧枪2确认"
   "Tag_15" := "拧紧枪2确认";
   IF #_w1 OR (("SERVER".设备状态2 = 20) AND ("SERVER".产品标识 = 538)) THEN "SERVER".设备状态2 := 21; END_IF;
END_REGION

REGION Network 23
   #IEC_Timer_0_Instance_17(IN := "SERVER".设备状态2 = 31, PT := T#5ms);   // TON
   #_w1 := #IEC_Timer_0_Instance_17.Q AND "拧紧枪3" AND NOT "Tag_30";   // rising edge of "拧紧枪3"
   "Tag_30" := "拧紧枪3";
   #IEC_Timer_0_Instance_18(IN := "SERVER".设备状态2 = 33, PT := T#5ms);   // TON
   #_w2 := #IEC_Timer_0_Instance_18.Q AND "拧紧枪3" AND NOT "Tag_60";   // rising edge of "拧紧枪3"
   "Tag_60" := "拧紧枪3";
   #IEC_Timer_0_Instance_19(IN := "SERVER".设备状态2 = 35, PT := T#5ms);   // TON
   #_w3 := #IEC_Timer_0_Instance_19.Q AND "拧紧枪3" AND NOT "Tag_61";   // rising edge of "拧紧枪3"
   "Tag_61" := "拧紧枪3";
   IF #_w1 OR (#IEC_Timer_0_Instance_17.Q AND NOT "控制器安装螺栓1") OR #_w2 OR (#IEC_Timer_0_Instance_18.Q AND NOT "控制器安装螺栓2") OR #_w3 OR (#IEC_Timer_0_Instance_19.Q AND NOT "控制器安装螺栓3") THEN
       "SERVER".设备状态2 := "SERVER".设备状态2 + 1;
   END_IF;
END_REGION

REGION Network 24
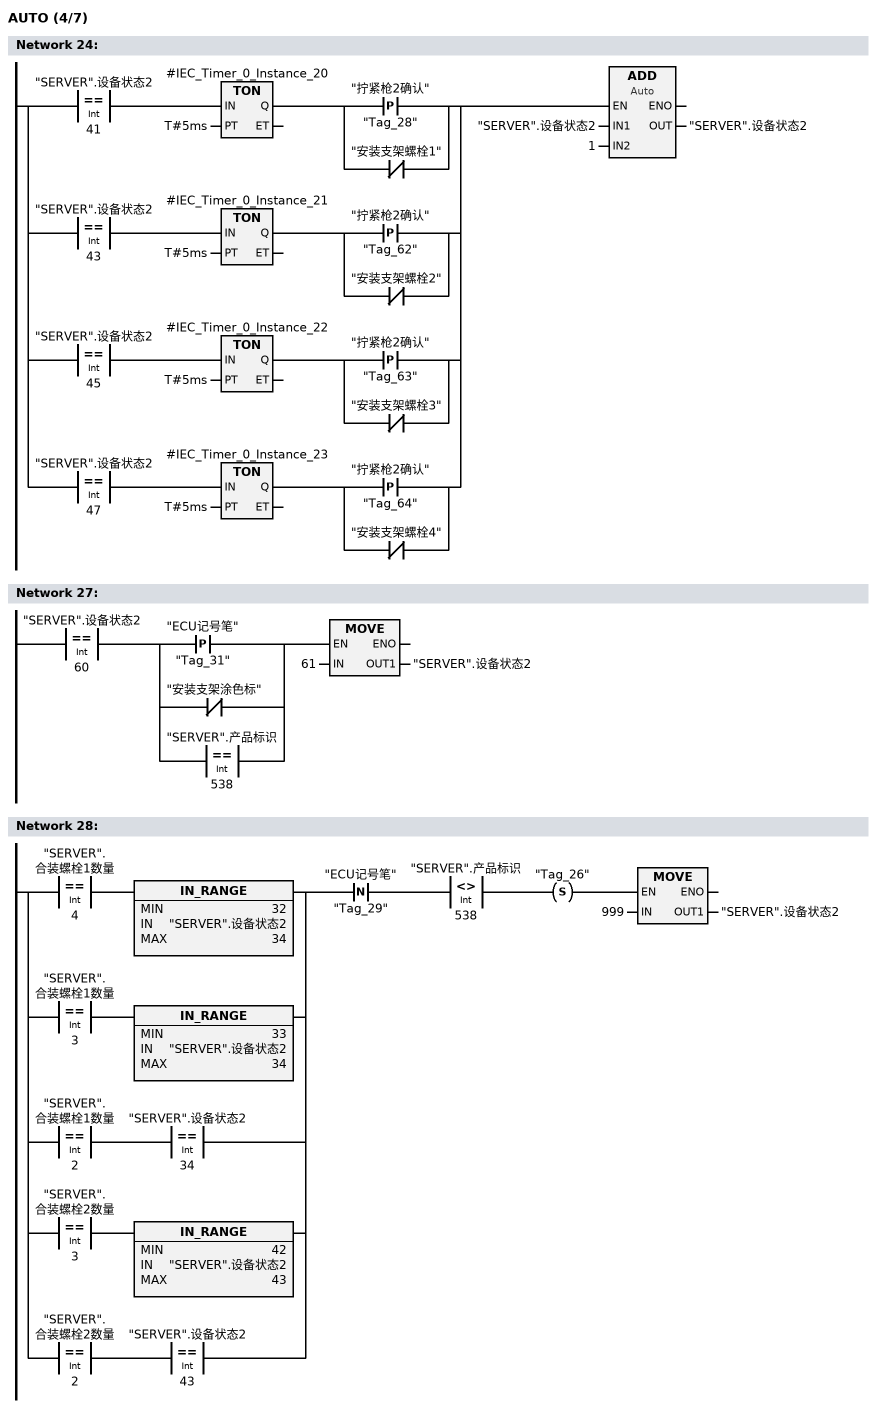
   #IEC_Timer_0_Instance_20(IN := "SERVER".设备状态2 = 41, PT := T#5ms);   // TON
   #_w1 := #IEC_Timer_0_Instance_20.Q AND "拧紧枪2确认" AND NOT "Tag_28";   // rising edge of "拧紧枪2确认"
   "Tag_28" := "拧紧枪2确认";
   #IEC_Timer_0_Instance_21(IN := "SERVER".设备状态2 = 43, PT := T#5ms);   // TON
   #_w2 := #IEC_Timer_0_Instance_21.Q AND "拧紧枪2确认" AND NOT "Tag_62";   // rising edge of "拧紧枪2确认"
   "Tag_62" := "拧紧枪2确认";
   #IEC_Timer_0_Instance_22(IN := "SERVER".设备状态2 = 45, PT := T#5ms);   // TON
   #_w3 := #IEC_Timer_0_Instance_22.Q AND "拧紧枪2确认" AND NOT "Tag_63";   // rising edge of "拧紧枪2确认"
   "Tag_63" := "拧紧枪2确认";
   #IEC_Timer_0_Instance_23(IN := "SERVER".设备状态2 = 47, PT := T#5ms);   // TON
   #_w4 := #IEC_Timer_0_Instance_23.Q AND "拧紧枪2确认" AND NOT "Tag_64";   // rising edge of "拧紧枪2确认"
   "Tag_64" := "拧紧枪2确认";
   IF #_w1 OR (#IEC_Timer_0_Instance_20.Q AND NOT "安装支架螺栓1") OR #_w2 OR (#IEC_Timer_0_Instance_21.Q AND NOT "安装支架螺栓2") OR #_w3 OR (#IEC_Timer_0_Instance_22.Q AND NOT "安装支架螺栓3") OR #_w4 OR (#IEC_Timer_0_Instance_23.Q AND NOT "安装支架螺栓4") THEN
       "SERVER".设备状态2 := "SERVER".设备状态2 + 1;
   END_IF;
END_REGION

REGION Network 27
   RUNG wire#powerrail
      { S7_Templates := "SrcType := Int" } EQ_Contact(in1 := "SERVER".设备状态2, in2 := 60)
      wire#w1
      P_Contact(operand := "ECU记号笔", bit := "Tag_31")
      wire#w2
      Move(in := 61, out1 => "SERVER".设备状态2)
   END_RUNG
   RUNG wire#w1
      I_Contact( "安装支架涂色标" )
   END_RUNG wire#w2
   RUNG wire#w1
      { S7_Templates := "SrcType := Int" } EQ_Contact(in1 := "SERVER".产品标识, in2 := 538)
   END_RUNG wire#w2
   // the same network as SCL:
   #_w1 := ("SERVER".设备状态2 = 60) AND "ECU记号笔" AND NOT "Tag_31";   // rising edge of "ECU记号笔"
   "Tag_31" := "ECU记号笔";
   IF #_w1 OR (("SERVER".设备状态2 = 60) AND (NOT "安装支架涂色标" OR ("SERVER".产品标识 = 538))) THEN
       "SERVER".设备状态2 := 61;
   END_IF;
END_REGION

REGION Network 28
   RUNG wire#powerrail
      { S7_Templates := "SrcType := Int" } EQ_Contact(in1 := "SERVER".合装螺栓1数量, in2 := 4)
      { S7_Templates := "SrcType := Int" } InRange(min := 32, in := "SERVER".设备状态2, max := 34)
      wire#w1
      N_Contact(operand := "ECU记号笔", bit := "Tag_29")
      { S7_Templates := "SrcType := Int" } NE_Contact(in1 := "SERVER".产品标识, in2 := 538)
      S_Coil( "Tag_26" )
      Move(in := 999, out1 => "SERVER".设备状态2)
   END_RUNG
   RUNG wire#powerrail
      { S7_Templates := "SrcType := Int" } EQ_Contact(in1 := "SERVER".合装螺栓1数量, in2 := 3)
      { S7_Templates := "SrcType := Int" } InRange(min := 33, in := "SERVER".设备状态2, max := 34)
   END_RUNG wire#w1
   RUNG wire#powerrail
      { S7_Templates := "SrcType := Int" } EQ_Contact(in1 := "SERVER".合装螺栓1数量, in2 := 2)
      { S7_Templates := "SrcType := Int" } EQ_Contact(in1 := "SERVER".设备状态2, in2 := 34)
   END_RUNG wire#w1
   RUNG wire#powerrail
      { S7_Templates := "SrcType := Int" } EQ_Contact(in1 := "SERVER".合装螺栓2数量, in2 := 3)
      { S7_Templates := "SrcType := Int" } InRange(min := 42, in := "SERVER".设备状态2, max := 43)
   END_RUNG wire#w1
   RUNG wire#powerrail
      { S7_Templates := "SrcType := Int" } EQ_Contact(in1 := "SERVER".合装螺栓2数量, in2 := 2)
      { S7_Templates := "SrcType := Int" } EQ_Contact(in1 := "SERVER".设备状态2, in2 := 43)
   END_RUNG wire#w1
   // the same network as SCL:
   #_w1 := ((("SERVER".合装螺栓1数量 = 4) AND (32 <= "SERVER".设备状态2) AND ("SERVER".设备状态2 <= 34)) OR (("SERVER".合装螺栓1数量 = 3) AND (33 <= "SERVER".设备状态2) AND ("SERVER".设备状态2 <= 34)) OR (("SERVER".合装螺栓1数量 = 2) AND ("SERVER".设备状态2 = 34)) OR (("SERVER".合装螺栓2数量 = 3) AND (42 <= "SERVER".设备状态2) AND ("SERVER".设备状态2 <= 43)) OR (("SERVER".合装螺栓2数量 = 2) AND ("SERVER".设备状态2 = 43))) AND NOT "ECU记号笔" AND "Tag_29";   // falling edge of "ECU记号笔"
   "Tag_29" := "ECU记号笔";
   IF #_w1 AND ("SERVER".产品标识 <> 538) THEN
       "Tag_26" := TRUE;
       "SERVER".设备状态2 := 999;
   END_IF;
END_REGION

REGION Network 29
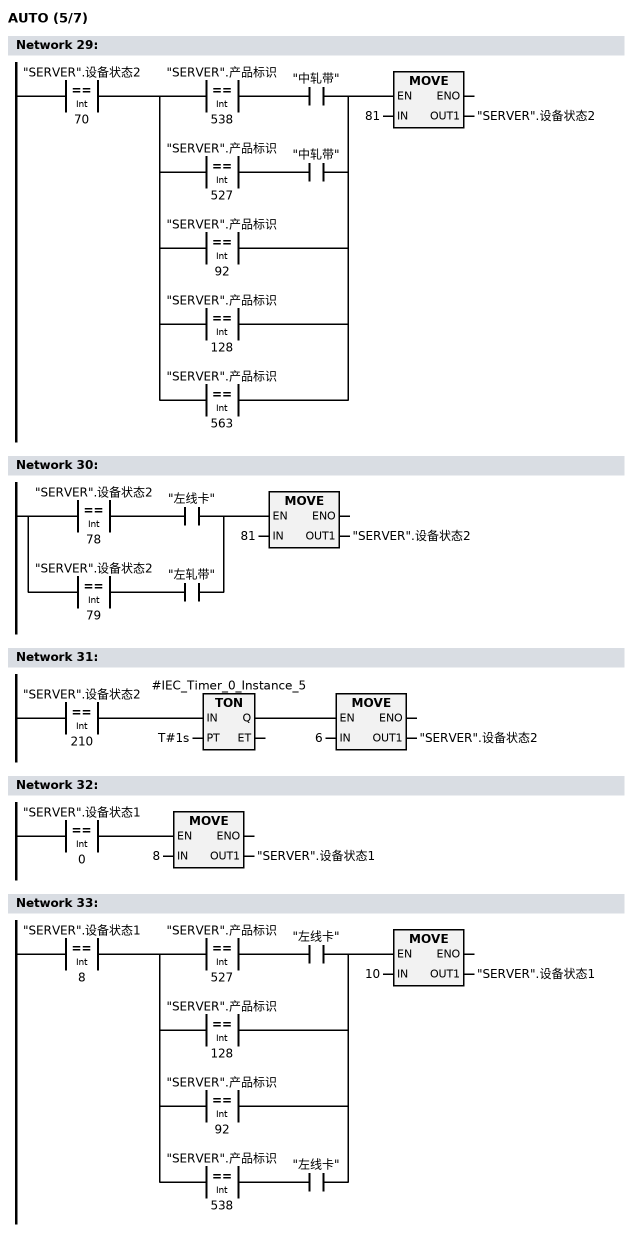
   RUNG wire#powerrail
      { S7_Templates := "SrcType := Int" } EQ_Contact(in1 := "SERVER".设备状态2, in2 := 70)
      wire#w1
      { S7_Templates := "SrcType := Int" } EQ_Contact(in1 := "SERVER".产品标识, in2 := 538)
      Contact( "中轧带" )
      wire#w2
      Move(in := 81, out1 => "SERVER".设备状态2)
   END_RUNG
   RUNG wire#w1
      { S7_Templates := "SrcType := Int" } EQ_Contact(in1 := "SERVER".产品标识, in2 := 527)
      Contact( "中轧带" )
   END_RUNG wire#w2
   RUNG wire#w1
      { S7_Templates := "SrcType := Int" } EQ_Contact(in1 := "SERVER".产品标识, in2 := 92)
   END_RUNG wire#w2
   RUNG wire#w1
      { S7_Templates := "SrcType := Int" } EQ_Contact(in1 := "SERVER".产品标识, in2 := 128)
   END_RUNG wire#w2
   RUNG wire#w1
      { S7_Templates := "SrcType := Int" } EQ_Contact(in1 := "SERVER".产品标识, in2 := 563)
   END_RUNG wire#w2
   // the same network as SCL:
   IF ("SERVER".设备状态2 = 70) AND ((("SERVER".产品标识 = 538) AND "中轧带") OR (("SERVER".产品标识 = 527) AND "中轧带") OR ("SERVER".产品标识 = 92) OR ("SERVER".产品标识 = 128) OR ("SERVER".产品标识 = 563)) THEN
       "SERVER".设备状态2 := 81;
   END_IF;
END_REGION

REGION Network 30
   RUNG wire#powerrail
      { S7_Templates := "SrcType := Int" } EQ_Contact(in1 := "SERVER".设备状态2, in2 := 78)
      Contact( "左线卡" )
      wire#w1
      Move(in := 81, out1 => "SERVER".设备状态2)
   END_RUNG
   RUNG wire#powerrail
      { S7_Templates := "SrcType := Int" } EQ_Contact(in1 := "SERVER".设备状态2, in2 := 79)
      Contact( "左轧带" )
   END_RUNG wire#w1
   // the same network as SCL:
   IF (("SERVER".设备状态2 = 78) AND "左线卡") OR (("SERVER".设备状态2 = 79) AND "左轧带") THEN
       "SERVER".设备状态2 := 81;
   END_IF;
END_REGION

REGION Network 31
   #IEC_Timer_0_Instance_5(IN := "SERVER".设备状态2 = 210, PT := T#1s);   // TON
   IF #IEC_Timer_0_Instance_5.Q THEN "SERVER".设备状态2 := 6; END_IF;
END_REGION

REGION Network 32
   RUNG wire#powerrail
      { S7_Templates := "SrcType := Int" } EQ_Contact(in1 := "SERVER".设备状态1, in2 := 0)
      Move(in := 8, out1 => "SERVER".设备状态1)
   END_RUNG
   // the same network as SCL:
   IF "SERVER".设备状态1 = 0 THEN "SERVER".设备状态1 := 8; END_IF;
END_REGION

REGION Network 33
   RUNG wire#powerrail
      { S7_Templates := "SrcType := Int" } EQ_Contact(in1 := "SERVER".设备状态1, in2 := 8)
      wire#w1
      { S7_Templates := "SrcType := Int" } EQ_Contact(in1 := "SERVER".产品标识, in2 := 527)
      Contact( "左线卡" )
      wire#w2
      Move(in := 10, out1 => "SERVER".设备状态1)
   END_RUNG
   RUNG wire#w1
      { S7_Templates := "SrcType := Int" } EQ_Contact(in1 := "SERVER".产品标识, in2 := 128)
   END_RUNG wire#w2
   RUNG wire#w1
      { S7_Templates := "SrcType := Int" } EQ_Contact(in1 := "SERVER".产品标识, in2 := 92)
   END_RUNG wire#w2
   RUNG wire#w1
      { S7_Templates := "SrcType := Int" } EQ_Contact(in1 := "SERVER".产品标识, in2 := 538)
      Contact( "左线卡" )
   END_RUNG wire#w2
   // the same network as SCL:
   IF ("SERVER".设备状态1 = 8) AND ((("SERVER".产品标识 = 527) AND "左线卡") OR ("SERVER".产品标识 = 128) OR ("SERVER".产品标识 = 92) OR (("SERVER".产品标识 = 538) AND "左线卡")) THEN
       "SERVER".设备状态1 := 10;
   END_IF;
END_REGION

REGION Network 34
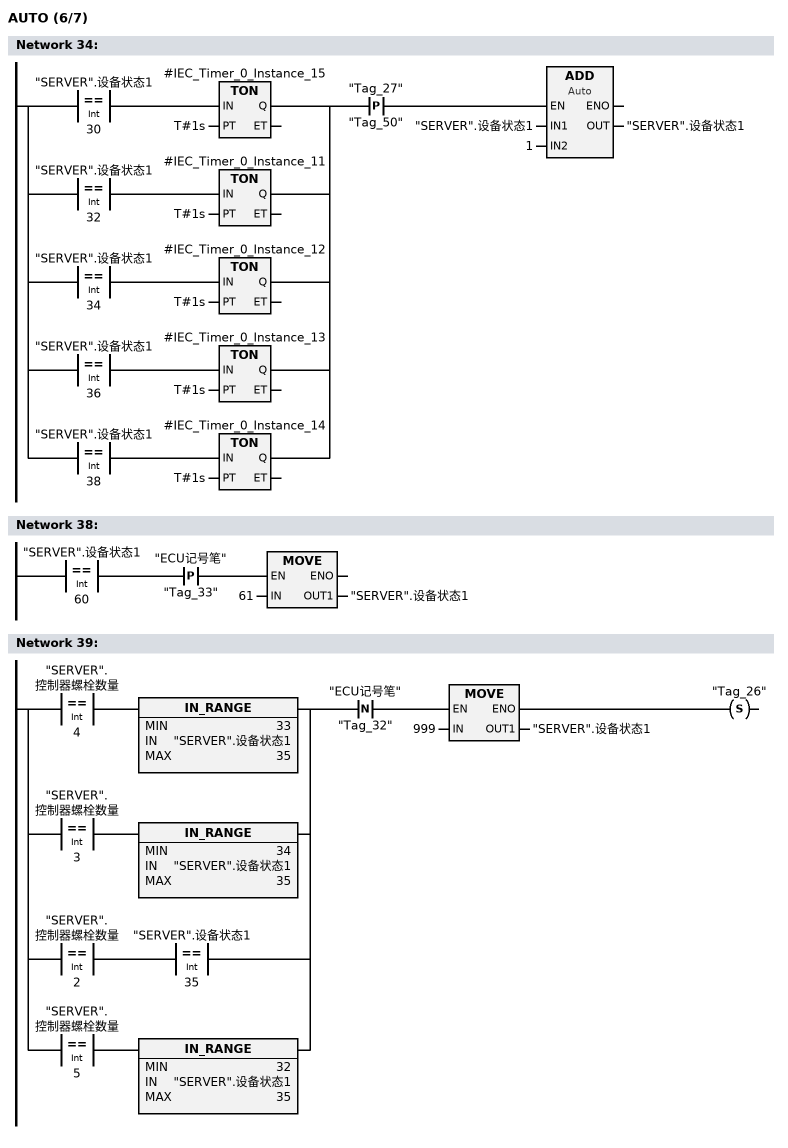
   #IEC_Timer_0_Instance_15(IN := "SERVER".设备状态1 = 30, PT := T#1s);   // TON
   #IEC_Timer_0_Instance_11(IN := "SERVER".设备状态1 = 32, PT := T#1s);   // TON
   #IEC_Timer_0_Instance_12(IN := "SERVER".设备状态1 = 34, PT := T#1s);   // TON
   #IEC_Timer_0_Instance_13(IN := "SERVER".设备状态1 = 36, PT := T#1s);   // TON
   #IEC_Timer_0_Instance_14(IN := "SERVER".设备状态1 = 38, PT := T#1s);   // TON
   #_w1 := (#IEC_Timer_0_Instance_15.Q OR #IEC_Timer_0_Instance_11.Q OR #IEC_Timer_0_Instance_12.Q OR #IEC_Timer_0_Instance_13.Q OR #IEC_Timer_0_Instance_14.Q) AND "Tag_27" AND NOT "Tag_50";   // rising edge of "Tag_27"
   "Tag_50" := "Tag_27";
   IF #_w1 THEN "SERVER".设备状态1 := "SERVER".设备状态1 + 1; END_IF;
END_REGION

REGION Network 38
   RUNG wire#powerrail
      { S7_Templates := "SrcType := Int" } EQ_Contact(in1 := "SERVER".设备状态1, in2 := 60)
      P_Contact(operand := "ECU记号笔", bit := "Tag_33")
      Move(in := 61, out1 => "SERVER".设备状态1)
   END_RUNG
   // the same network as SCL:
   #_w1 := ("SERVER".设备状态1 = 60) AND "ECU记号笔" AND NOT "Tag_33";   // rising edge of "ECU记号笔"
   "Tag_33" := "ECU记号笔";
   IF #_w1 THEN "SERVER".设备状态1 := 61; END_IF;
END_REGION

REGION Network 39
   RUNG wire#powerrail
      { S7_Templates := "SrcType := Int" } EQ_Contact(in1 := "SERVER".控制器螺栓数量, in2 := 4)
      { S7_Templates := "SrcType := Int" } InRange(min := 33, in := "SERVER".设备状态1, max := 35)
      wire#w1
      N_Contact(operand := "ECU记号笔", bit := "Tag_32")
      Move(in := 999, out1 => "SERVER".设备状态1)
      S_Coil( "Tag_26" )
   END_RUNG
   RUNG wire#powerrail
      { S7_Templates := "SrcType := Int" } EQ_Contact(in1 := "SERVER".控制器螺栓数量, in2 := 3)
      { S7_Templates := "SrcType := Int" } InRange(min := 34, in := "SERVER".设备状态1, max := 35)
   END_RUNG wire#w1
   RUNG wire#powerrail
      { S7_Templates := "SrcType := Int" } EQ_Contact(in1 := "SERVER".控制器螺栓数量, in2 := 2)
      { S7_Templates := "SrcType := Int" } EQ_Contact(in1 := "SERVER".设备状态1, in2 := 35)
   END_RUNG wire#w1
   RUNG wire#powerrail
      { S7_Templates := "SrcType := Int" } EQ_Contact(in1 := "SERVER".控制器螺栓数量, in2 := 5)
      { S7_Templates := "SrcType := Int" } InRange(min := 32, in := "SERVER".设备状态1, max := 35)
   END_RUNG wire#w1
   // the same network as SCL:
   #_w1 := ((("SERVER".控制器螺栓数量 = 4) AND (33 <= "SERVER".设备状态1) AND ("SERVER".设备状态1 <= 35)) OR (("SERVER".控制器螺栓数量 = 3) AND (34 <= "SERVER".设备状态1) AND ("SERVER".设备状态1 <= 35)) OR (("SERVER".控制器螺栓数量 = 2) AND ("SERVER".设备状态1 = 35)) OR (("SERVER".控制器螺栓数量 = 5) AND (32 <= "SERVER".设备状态1) AND ("SERVER".设备状态1 <= 35))) AND NOT "ECU记号笔" AND "Tag_32";   // falling edge of "ECU记号笔"
   "Tag_32" := "ECU记号笔";
   IF #_w1 THEN
       "SERVER".设备状态1 := 999;
       "Tag_26" := TRUE;
   END_IF;
END_REGION

REGION Network 40
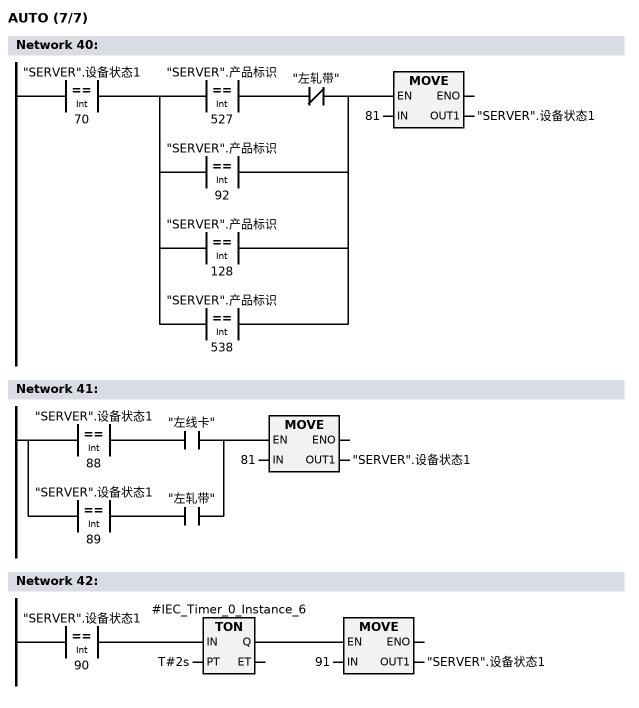
   RUNG wire#powerrail
      { S7_Templates := "SrcType := Int" } EQ_Contact(in1 := "SERVER".设备状态1, in2 := 70)
      wire#w1
      { S7_Templates := "SrcType := Int" } EQ_Contact(in1 := "SERVER".产品标识, in2 := 527)
      I_Contact( "左轧带" )
      wire#w2
      Move(in := 81, out1 => "SERVER".设备状态1)
   END_RUNG
   RUNG wire#w1
      { S7_Templates := "SrcType := Int" } EQ_Contact(in1 := "SERVER".产品标识, in2 := 92)
   END_RUNG wire#w2
   RUNG wire#w1
      { S7_Templates := "SrcType := Int" } EQ_Contact(in1 := "SERVER".产品标识, in2 := 128)
   END_RUNG wire#w2
   RUNG wire#w1
      { S7_Templates := "SrcType := Int" } EQ_Contact(in1 := "SERVER".产品标识, in2 := 538)
   END_RUNG wire#w2
   // the same network as SCL:
   IF ("SERVER".设备状态1 = 70) AND ((("SERVER".产品标识 = 527) AND NOT "左轧带") OR ("SERVER".产品标识 = 92) OR ("SERVER".产品标识 = 128) OR ("SERVER".产品标识 = 538)) THEN
       "SERVER".设备状态1 := 81;
   END_IF;
END_REGION

REGION Network 41
   RUNG wire#powerrail
      { S7_Templates := "SrcType := Int" } EQ_Contact(in1 := "SERVER".设备状态1, in2 := 88)
      Contact( "左线卡" )
      wire#w1
      Move(in := 81, out1 => "SERVER".设备状态1)
   END_RUNG
   RUNG wire#powerrail
      { S7_Templates := "SrcType := Int" } EQ_Contact(in1 := "SERVER".设备状态1, in2 := 89)
      Contact( "左轧带" )
   END_RUNG wire#w1
   // the same network as SCL:
   IF (("SERVER".设备状态1 = 88) AND "左线卡") OR (("SERVER".设备状态1 = 89) AND "左轧带") THEN
       "SERVER".设备状态1 := 81;
   END_IF;
END_REGION

REGION Network 42
   #IEC_Timer_0_Instance_6(IN := "SERVER".设备状态1 = 90, PT := T#2s);   // TON
   IF #IEC_Timer_0_Instance_6.Q THEN "SERVER".设备状态1 := 91; END_IF;
END_REGION
END_FUNCTION_BLOCK

FUNCTION_BLOCK "CCD检测"   // FB5, LAD
{ S7_Optimized_Access := 'TRUE' }
VERSION : 0.1
   VAR_INPUT
      ccd_pro_start : Bool;
      "Command Number" : Int;
   END_VAR
   VAR_OUTPUT
      done : Bool;
   END_VAR
   VAR
      "step" : Int;
      PRO : Int;
      Chg_start : Bool;
      Chg_done : Bool;
      CCD_PRO_temp1 : Int;
      CCD_PRO_temp2 : Int;
      IEC_Timer_0_Instance : TON_TIME;
      IEC_Timer_0_Instance_1 : TON_TIME;
      IEC_Timer_0_Instance_2 : TON_TIME;
      IEC_Timer_0_Instance_3 : TON_TIME;
      IEC_Timer_0_Instance_4 : TON_TIME;
   END_VAR
   VAR_TEMP   // added for the SCL form of the ladder/FBD networks
      _w1 : Bool;
      _w2 : Bool;
   END_VAR
BEGIN

REGION Network 1
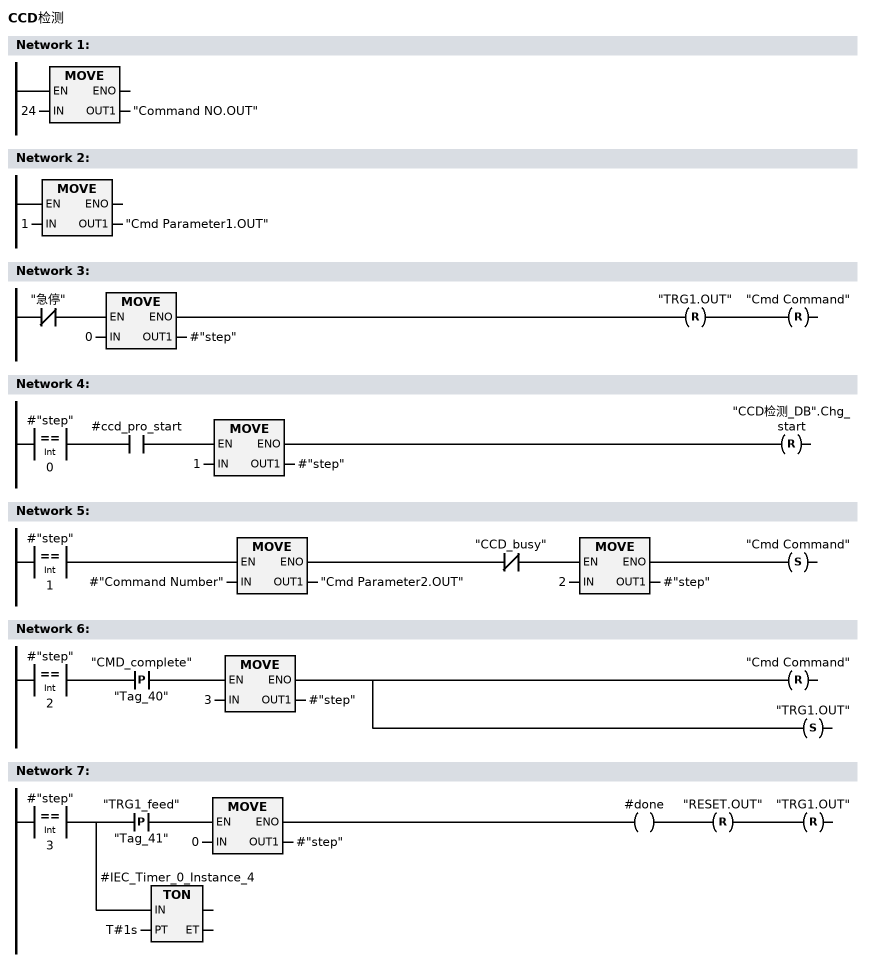
   RUNG wire#powerrail
      Move(in := 24, out1 => "Command NO.OUT")
   END_RUNG
   // the same network as SCL:
   "Command NO.OUT" := 24;
END_REGION

REGION Network 2
   RUNG wire#powerrail
      Move(in := 1, out1 => "Cmd Parameter1.OUT")
   END_RUNG
   // the same network as SCL:
   "Cmd Parameter1.OUT" := 1;
END_REGION

REGION Network 3
   RUNG wire#powerrail
      I_Contact( "急停" )
      Move(in := 0, out1 => #"step")
      R_Coil( "TRG1.OUT" )
      R_Coil( "Cmd Command" )
   END_RUNG
   // the same network as SCL:
   IF NOT "急停" THEN
       #"step" := 0;
       "TRG1.OUT" := FALSE;
       "Cmd Command" := FALSE;
   END_IF;
END_REGION

REGION Network 4
   RUNG wire#powerrail
      { S7_Templates := "SrcType := Int" } EQ_Contact(in1 := #"step", in2 := 0)
      Contact( #ccd_pro_start )
      Move(in := 1, out1 => #"step")
      R_Coil( "CCD检测_DB".Chg_start )
   END_RUNG
   // the same network as SCL:
   #_w1 := (#"step" = 0) AND #ccd_pro_start;
   IF #_w1 THEN
       #"step" := 1;
       "CCD检测_DB".Chg_start := FALSE;
   END_IF;
END_REGION

REGION Network 5
   RUNG wire#powerrail
      { S7_Templates := "SrcType := Int" } EQ_Contact(in1 := #"step", in2 := 1)
      Move(in := #"Command Number", out1 => "Cmd Parameter2.OUT")
      I_Contact( "CCD_busy" )
      Move(in := 2, out1 => #"step")
      S_Coil( "Cmd Command" )
   END_RUNG
   // the same network as SCL:
   #_w1 := #"step" = 1;
   IF #_w1 THEN "Cmd Parameter2.OUT" := #"Command Number"; END_IF;
   IF #_w1 AND NOT "CCD_busy" THEN
       #"step" := 2;
       "Cmd Command" := TRUE;
   END_IF;
END_REGION

REGION Network 6
   RUNG wire#powerrail
      { S7_Templates := "SrcType := Int" } EQ_Contact(in1 := #"step", in2 := 2)
      P_Contact(operand := "CMD_complete", bit := "Tag_40")
      Move(in := 3, out1 => #"step")
      wire#w1
      R_Coil( "Cmd Command" )
   END_RUNG
   RUNG wire#w1
      S_Coil( "TRG1.OUT" )
   END_RUNG
   // the same network as SCL:
   #_w1 := (#"step" = 2) AND "CMD_complete" AND NOT "Tag_40";   // rising edge of "CMD_complete"
   "Tag_40" := "CMD_complete";
   IF #_w1 THEN
       #"step" := 3;
       "Cmd Command" := FALSE;
       "TRG1.OUT" := TRUE;
   END_IF;
END_REGION

REGION Network 7
   #_w1 := #"step" = 3;
   #_w2 := #_w1 AND "TRG1_feed" AND NOT "Tag_41";   // rising edge of "TRG1_feed"
   "Tag_41" := "TRG1_feed";
   IF #_w2 THEN #"step" := 0; END_IF;
   #done := #_w2;
   IF #_w2 THEN
       "RESET.OUT" := FALSE;
       "TRG1.OUT" := FALSE;
   END_IF;
   #IEC_Timer_0_Instance_4(IN := #_w1, PT := T#1s);   // TON
END_REGION
END_FUNCTION_BLOCK

ORGANIZATION_BLOCK "Main"   // OB1, LAD, ProgramCycle
TITLE = "Main Program Sweep (Cycle)"
{ S7_Optimized_Access := 'TRUE' }
VERSION : 0.1
   VAR_INPUT
      Initial_Call : Bool;   // Initial call of this OB
      Remanence : Bool;   // =True, if remanent data are available
   END_VAR
   VAR_TEMP   // added for the SCL form of the ladder/FBD networks
      _w1 : Bool;
   END_VAR
BEGIN

REGION Network 1
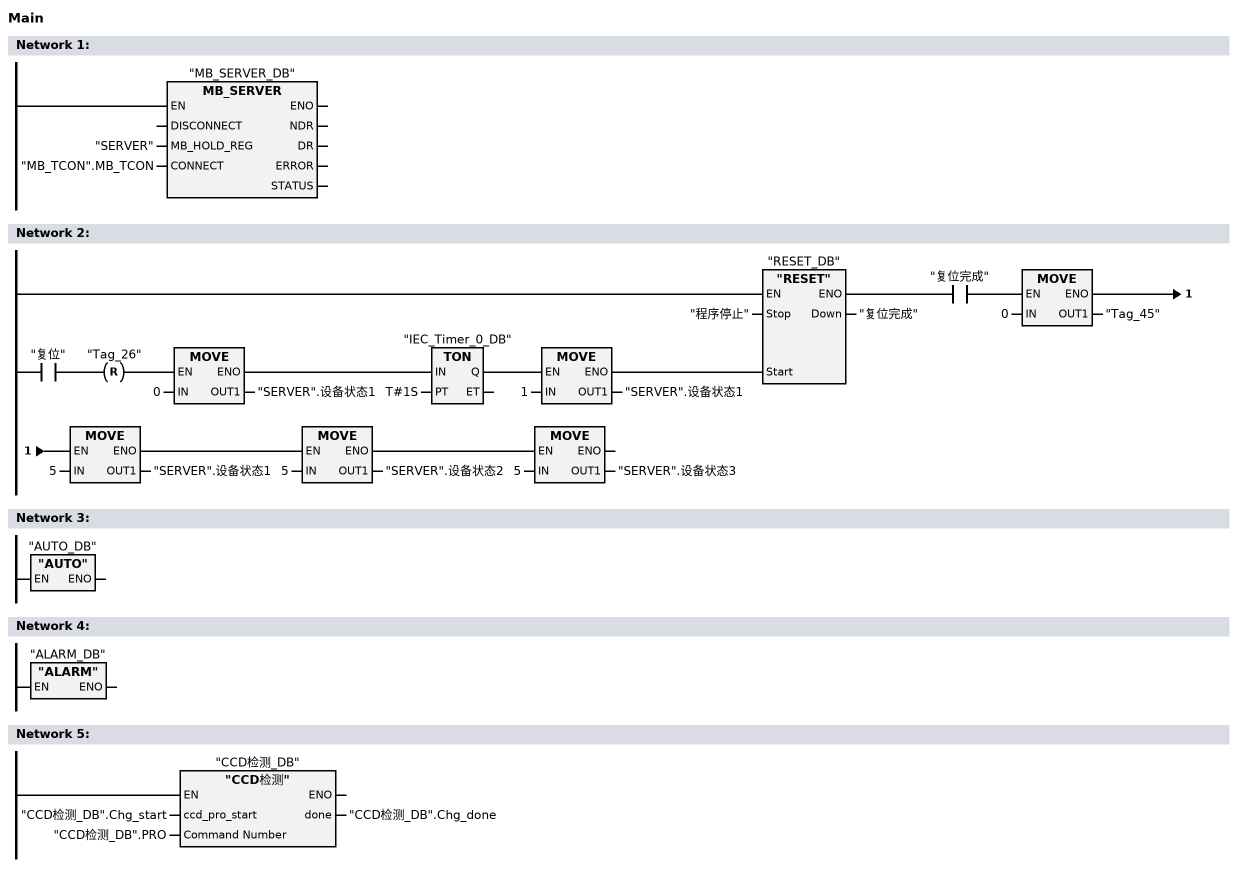
   "MB_SERVER_DB"(MB_HOLD_REG := "SERVER", CONNECT := "MB_TCON".MB_TCON);   // MB_SERVER
END_REGION

REGION Network 2
   IF "复位" THEN
       "Tag_26" := FALSE;
       "SERVER".设备状态1 := 0;
   END_IF;
   "IEC_Timer_0_DB".TON(IN := "复位", PT := T#1S);
   IF "IEC_Timer_0_DB".Q THEN "SERVER".设备状态1 := 1; END_IF;
   "RESET_DB"(Stop := "程序停止", Start := "IEC_Timer_0_DB".Q, Down => "复位完成", ENO => #_w1);   // "RESET"
   IF #_w1 AND "复位完成" THEN
       "Tag_45" := 0;
       "SERVER".设备状态1 := 5;
       "SERVER".设备状态2 := 5;
       "SERVER".设备状态3 := 5;
   END_IF;
END_REGION

REGION Network 3
   RUNG wire#powerrail
      "AUTO_DB"()
   END_RUNG
   // the same network as SCL:
   "AUTO_DB"();   // "AUTO"
END_REGION

REGION Network 4
   RUNG wire#powerrail
      "ALARM_DB"()
   END_RUNG
   // the same network as SCL:
   "ALARM_DB"();   // "ALARM"
END_REGION

REGION Network 5
   RUNG wire#powerrail
      "CCD检测_DB"(ccd_pro_start := "CCD检测_DB".Chg_start, "Command Number" := "CCD检测_DB".PRO, done => "CCD检测_DB".Chg_done)
   END_RUNG
   // the same network as SCL:
   "CCD检测_DB"(ccd_pro_start := "CCD检测_DB".Chg_start,   // "CCD检测"
              "Command Number" := "CCD检测_DB".PRO,
              done => "CCD检测_DB".Chg_done);
END_REGION
END_ORGANIZATION_BLOCK

ORGANIZATION_BLOCK "Cyclic interrupt_10ms"   // OB30, LAD, CyclicInterrupt
{ S7_Optimized_Access := 'TRUE' }
VERSION : 0.1
   VAR_INPUT
      Initial_Call : Bool;   // Initial call of this OB
      Event_Count : Int;   // Events discarded
   END_VAR
   VAR_TEMP
      done : Bool;
      done_1 : Bool;
      busy : Bool;
      direction : Bool;
      speed : Real;
      temp2 : Int;
      temp1 : Real;
      torque : Real;
   END_VAR
BEGIN

REGION Network 1
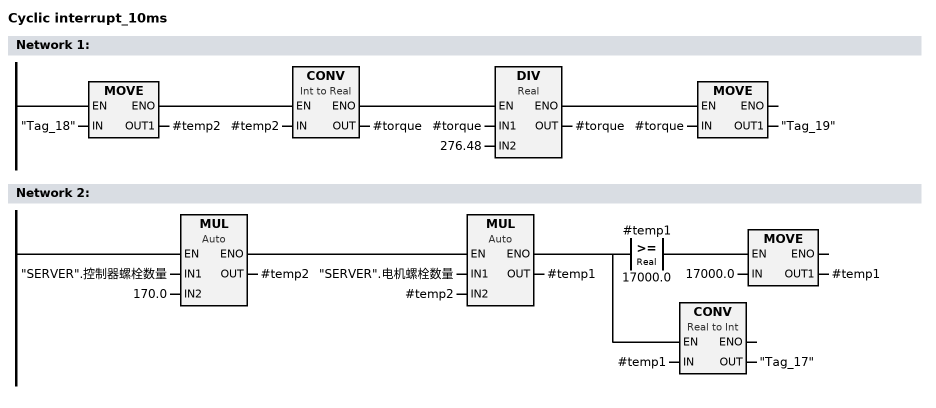
   RUNG wire#powerrail
      Move(in := "Tag_18", out1 => #temp2)
      { S7_Templates := "[SrcType := Int, DestType := Real]" } Convert(in := #temp2, out => #torque)
      { S7_Templates := "SrcType := Real" } Div(in1 := #torque, in2 := 276.48, out => #torque)
      Move(in := #torque, out1 => "Tag_19")
   END_RUNG
   // the same network as SCL:
   #temp2 := "Tag_18";
   #torque := INT_TO_REAL(#temp2);
   #torque := #torque / 276.48;
   "Tag_19" := #torque;
END_REGION

REGION Network 2
   RUNG wire#powerrail
      Mul(in1 := "SERVER".控制器螺栓数量, in2 := 170.0, out => #temp2)
      Mul(in1 := "SERVER".电机螺栓数量, in2 := #temp2, out => #temp1)
      wire#w1
      { S7_Templates := "SrcType := Real" } GE_Contact(in1 := #temp1, in2 := 17000.0)
      Move(in := 17000.0, out1 => #temp1)
   END_RUNG
   RUNG wire#w1
      { S7_Templates := "[SrcType := Real, DestType := Int]" } Convert(in := #temp1, out => "Tag_17")
   END_RUNG
   // the same network as SCL:
   #temp2 := "SERVER".控制器螺栓数量 * 170.0;
   #temp1 := "SERVER".电机螺栓数量 * #temp2;
   IF #temp1 >= 17000.0 THEN #temp1 := 17000.0; END_IF;
   "Tag_17" := REAL_TO_INT(#temp1);
END_REGION
END_ORGANIZATION_BLOCK